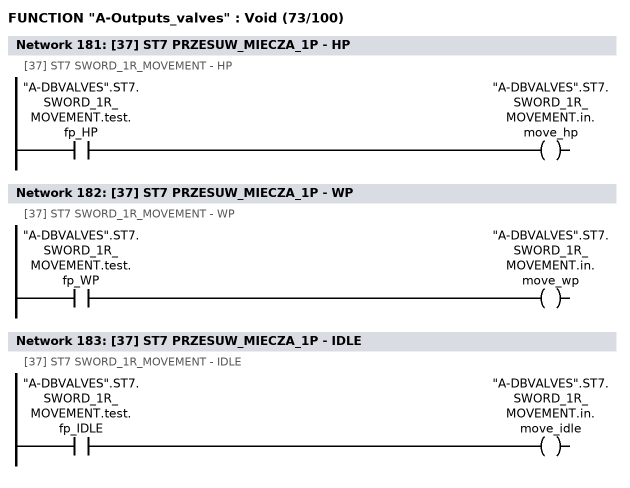
      O "A-DBVALVES".ST7.SWORD_1R_MOVEMENT.test.fp_HP;
//    O     "A-Flags".STATION.IN_HP_STEP
      = "A-DBVALVES".ST7.SWORD_1R_MOVEMENT.in.move_hp;
NETWORK
TITLE = [37] ST7 PRZESUW_MIECZA_1P - WP
//[37] ST7 SWORD_1R_MOVEMENT - WP
      O "A-DBVALVES".ST7.SWORD_1R_MOVEMENT.test.fp_WP;
      = "A-DBVALVES".ST7.SWORD_1R_MOVEMENT.in.move_wp;
NETWORK
TITLE = [37] ST7 PRZESUW_MIECZA_1P - IDLE
//[37] ST7 SWORD_1R_MOVEMENT - IDLE
      O "A-DBVALVES".ST7.SWORD_1R_MOVEMENT.test.fp_IDLE;
      = "A-DBVALVES".ST7.SWORD_1R_MOVEMENT.in.move_idle;
NETWORK
TITLE = [37] ST7 PRZESUW_MIECZA_1P
//[37] ST7 SWORD_1R_MOVEMENT
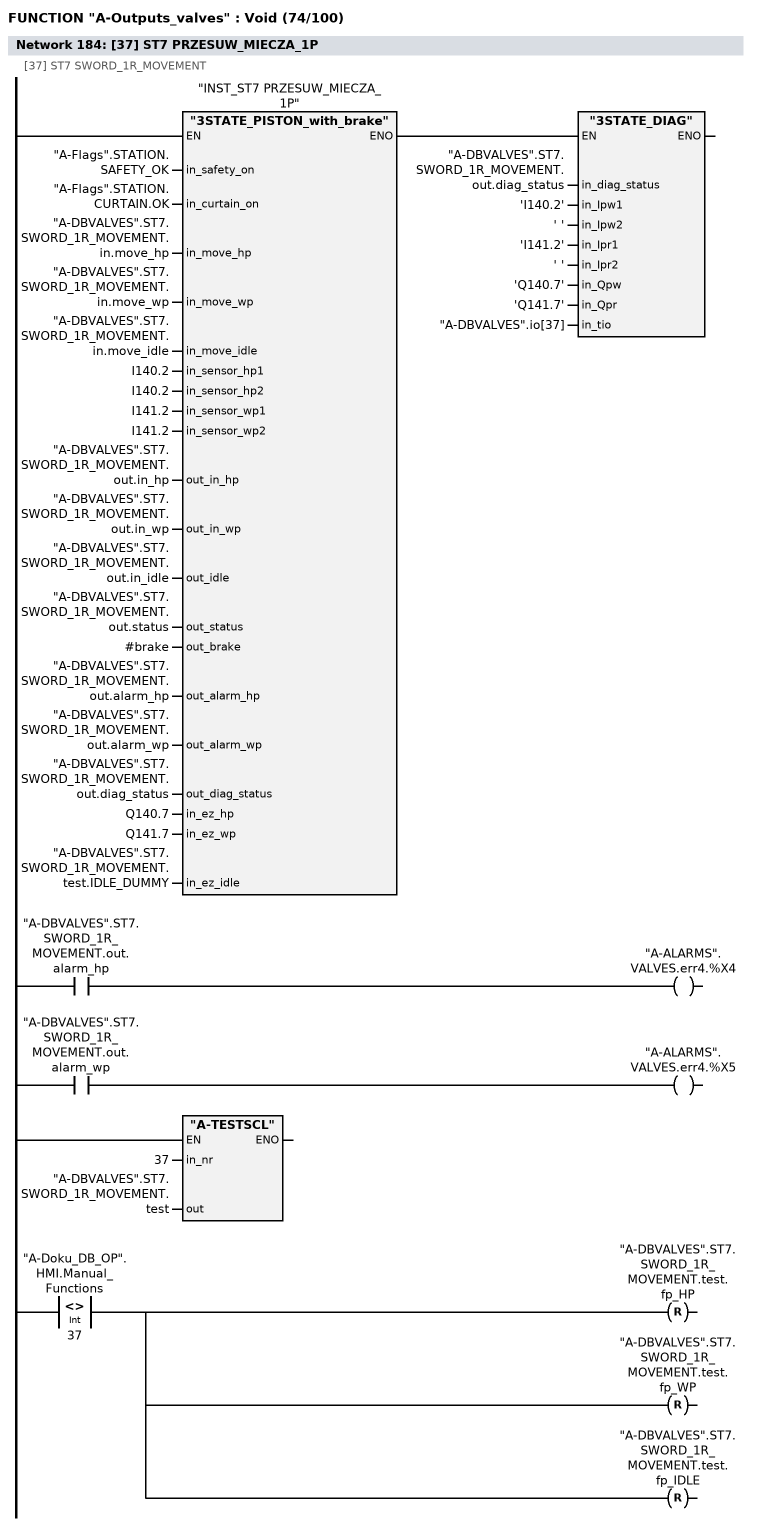
      CALL "3STATE_PISTON_with_brake", "INST_ST7 PRZESUW_MIECZA_1P"
      (  in_safety_on                := "A-Flags".STATION.SAFETY_OK ,
         in_curtain_on               := "A-Flags".STATION.CURTAIN.OK ,
         in_move_hp                  := "A-DBVALVES".ST7.SWORD_1R_MOVEMENT.in.move_hp ,
         in_move_wp                  := "A-DBVALVES".ST7.SWORD_1R_MOVEMENT.in.move_wp ,
         in_move_idle                := "A-DBVALVES".ST7.SWORD_1R_MOVEMENT.in.move_idle ,
         in_sensor_hp1               := I140.2 ,
         in_sensor_hp2               := I140.2 ,
         in_sensor_wp1               := I141.2 ,
         in_sensor_wp2               := I141.2 ,
         out_in_hp                   := "A-DBVALVES".ST7.SWORD_1R_MOVEMENT.out.in_hp ,
         out_in_wp                   := "A-DBVALVES".ST7.SWORD_1R_MOVEMENT.out.in_wp ,
         out_idle                    := "A-DBVALVES".ST7.SWORD_1R_MOVEMENT.out.in_idle ,
         out_status                  := "A-DBVALVES".ST7.SWORD_1R_MOVEMENT.out.status ,
         out_brake                   := #brake ,
         out_alarm_hp                := "A-DBVALVES".ST7.SWORD_1R_MOVEMENT.out.alarm_hp ,
         out_alarm_wp                := "A-DBVALVES".ST7.SWORD_1R_MOVEMENT.out.alarm_wp ,
         out_diag_status             := "A-DBVALVES".ST7.SWORD_1R_MOVEMENT.out.diag_status ,
         in_ez_hp                    := Q140.7 ,
         in_ez_wp                    := Q141.7 ,
         in_ez_idle                  := "A-DBVALVES".ST7.SWORD_1R_MOVEMENT.test.IDLE_DUMMY
      );

      CALL "3STATE_DIAG"
      (  in_diag_status              := "A-DBVALVES".ST7.SWORD_1R_MOVEMENT.out.diag_status ,
         in_Ipw1                     := 'I140.2' ,
         in_Ipw2                     := ' ' ,
         in_Ipr1                     := 'I141.2' ,
         in_Ipr2                     := ' ' ,
         in_Qpw                      := 'Q140.7' ,
         in_Qpr                      := 'Q141.7' ,
         in_tio                      := "A-DBVALVES".io[37]
      );

      A "A-DBVALVES".ST7.SWORD_1R_MOVEMENT.out.alarm_hp;
      = "A-ALARMS".VALVES.err4.%X4;

      A "A-DBVALVES".ST7.SWORD_1R_MOVEMENT.out.alarm_wp;
      = "A-ALARMS".VALVES.err4.%X5;

      CALL "A-TESTSCL"
      (  in_nr                       := 37 ,
         out                         := "A-DBVALVES".ST7.SWORD_1R_MOVEMENT.test
      );

      A(;
      L "A-Doku_DB_OP".HMI.Manual_Functions;
      L 37;
      <>I;
      );
      R "A-DBVALVES".ST7.SWORD_1R_MOVEMENT.test.fp_HP;
      R "A-DBVALVES".ST7.SWORD_1R_MOVEMENT.test.fp_WP;
      R "A-DBVALVES".ST7.SWORD_1R_MOVEMENT.test.fp_IDLE;
NETWORK
TITLE = -

NETWORK
TITLE = [38] ST7 PRZESUW_DOCISKOW - HP
//[38] ST7 HOLDFAST_MOVEMENT - HP
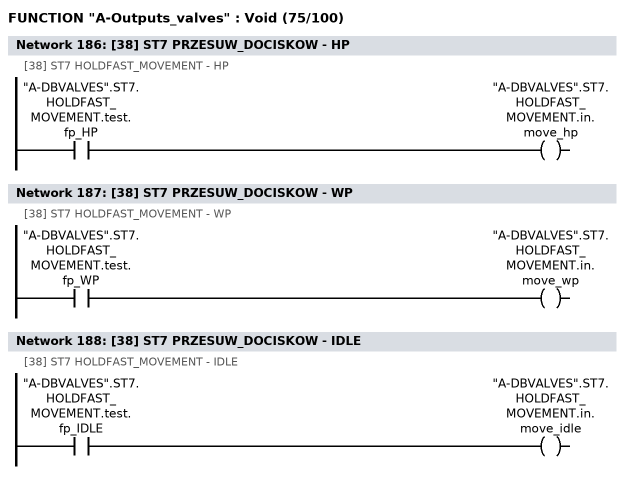
      O "A-DBVALVES".ST7.HOLDFAST_MOVEMENT.test.fp_HP;
//    O     "A-Flags".STATION.IN_HP_STEP
      = "A-DBVALVES".ST7.HOLDFAST_MOVEMENT.in.move_hp;
NETWORK
TITLE = [38] ST7 PRZESUW_DOCISKOW - WP
//[38] ST7 HOLDFAST_MOVEMENT - WP
      O "A-DBVALVES".ST7.HOLDFAST_MOVEMENT.test.fp_WP;
      = "A-DBVALVES".ST7.HOLDFAST_MOVEMENT.in.move_wp;
NETWORK
TITLE = [38] ST7 PRZESUW_DOCISKOW - IDLE
//[38] ST7 HOLDFAST_MOVEMENT - IDLE
      O "A-DBVALVES".ST7.HOLDFAST_MOVEMENT.test.fp_IDLE;
      = "A-DBVALVES".ST7.HOLDFAST_MOVEMENT.in.move_idle;
NETWORK
TITLE = [38] ST7 PRZESUW_DOCISKOW
//[38] ST7 HOLDFAST_MOVEMENT
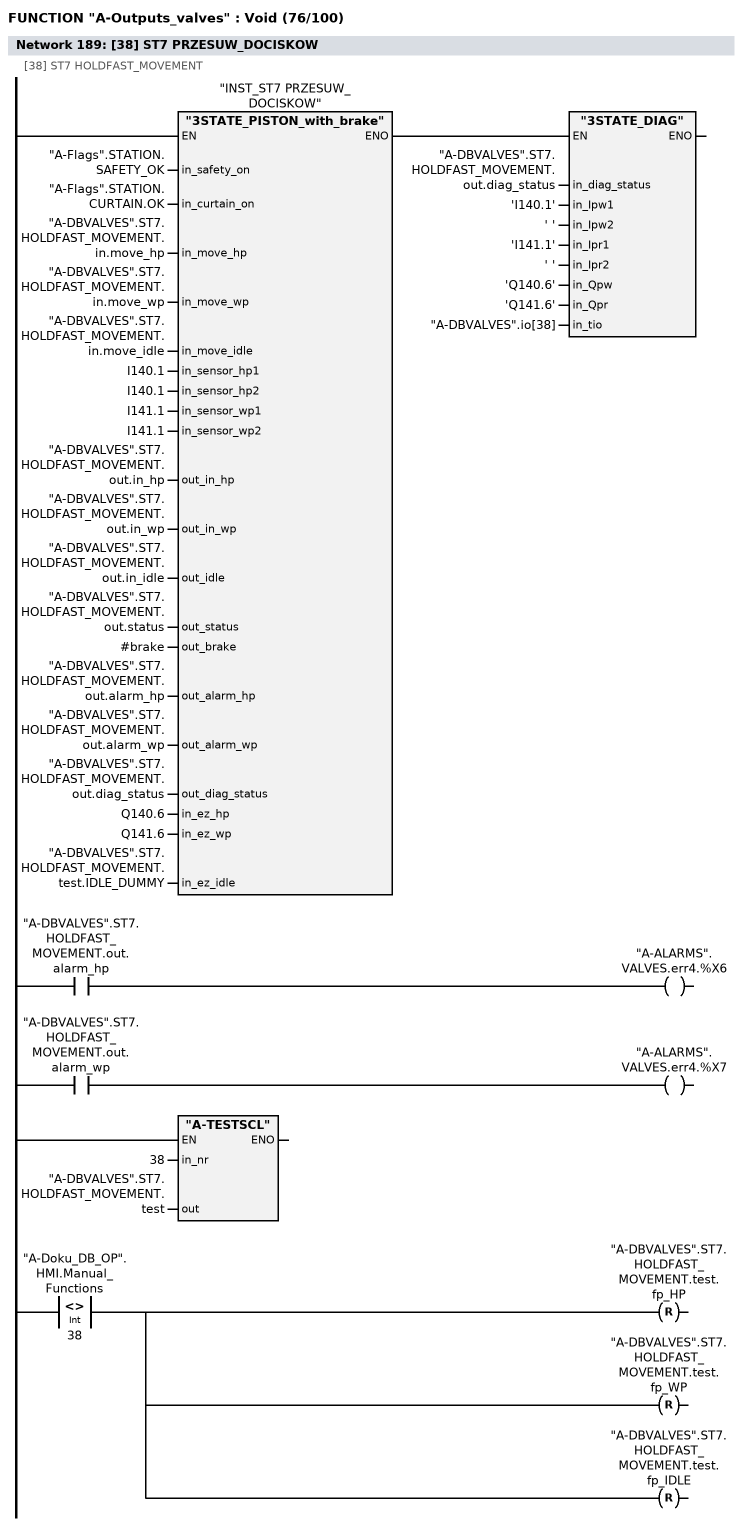
      CALL "3STATE_PISTON_with_brake", "INST_ST7 PRZESUW_DOCISKOW"
      (  in_safety_on                := "A-Flags".STATION.SAFETY_OK ,
         in_curtain_on               := "A-Flags".STATION.CURTAIN.OK ,
         in_move_hp                  := "A-DBVALVES".ST7.HOLDFAST_MOVEMENT.in.move_hp ,
         in_move_wp                  := "A-DBVALVES".ST7.HOLDFAST_MOVEMENT.in.move_wp ,
         in_move_idle                := "A-DBVALVES".ST7.HOLDFAST_MOVEMENT.in.move_idle ,
         in_sensor_hp1               := I140.1 ,
         in_sensor_hp2               := I140.1 ,
         in_sensor_wp1               := I141.1 ,
         in_sensor_wp2               := I141.1 ,
         out_in_hp                   := "A-DBVALVES".ST7.HOLDFAST_MOVEMENT.out.in_hp ,
         out_in_wp                   := "A-DBVALVES".ST7.HOLDFAST_MOVEMENT.out.in_wp ,
         out_idle                    := "A-DBVALVES".ST7.HOLDFAST_MOVEMENT.out.in_idle ,
         out_status                  := "A-DBVALVES".ST7.HOLDFAST_MOVEMENT.out.status ,
         out_brake                   := #brake ,
         out_alarm_hp                := "A-DBVALVES".ST7.HOLDFAST_MOVEMENT.out.alarm_hp ,
         out_alarm_wp                := "A-DBVALVES".ST7.HOLDFAST_MOVEMENT.out.alarm_wp ,
         out_diag_status             := "A-DBVALVES".ST7.HOLDFAST_MOVEMENT.out.diag_status ,
         in_ez_hp                    := Q140.6 ,
         in_ez_wp                    := Q141.6 ,
         in_ez_idle                  := "A-DBVALVES".ST7.HOLDFAST_MOVEMENT.test.IDLE_DUMMY
      );

      CALL "3STATE_DIAG"
      (  in_diag_status              := "A-DBVALVES".ST7.HOLDFAST_MOVEMENT.out.diag_status ,
         in_Ipw1                     := 'I140.1' ,
         in_Ipw2                     := ' ' ,
         in_Ipr1                     := 'I141.1' ,
         in_Ipr2                     := ' ' ,
         in_Qpw                      := 'Q140.6' ,
         in_Qpr                      := 'Q141.6' ,
         in_tio                      := "A-DBVALVES".io[38]
      );

      A "A-DBVALVES".ST7.HOLDFAST_MOVEMENT.out.alarm_hp;
      = "A-ALARMS".VALVES.err4.%X6;

      A "A-DBVALVES".ST7.HOLDFAST_MOVEMENT.out.alarm_wp;
      = "A-ALARMS".VALVES.err4.%X7;

      CALL "A-TESTSCL"
      (  in_nr                       := 38 ,
         out                         := "A-DBVALVES".ST7.HOLDFAST_MOVEMENT.test
      );

      A(;
      L "A-Doku_DB_OP".HMI.Manual_Functions;
      L 38;
      <>I;
      );
      R "A-DBVALVES".ST7.HOLDFAST_MOVEMENT.test.fp_HP;
      R "A-DBVALVES".ST7.HOLDFAST_MOVEMENT.test.fp_WP;
      R "A-DBVALVES".ST7.HOLDFAST_MOVEMENT.test.fp_IDLE;
NETWORK
TITLE = -

NETWORK
TITLE = [39] ST7 PRZESUW_MIECZA_Y_2L - HP
//[39] ST7 SWORD_Y_2L_MOVEMENT - HP
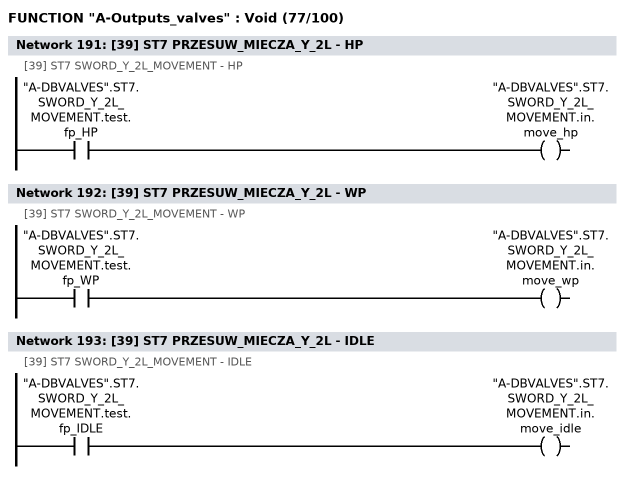
      O "A-DBVALVES".ST7.SWORD_Y_2L_MOVEMENT.test.fp_HP;
//    O     "A-Flags".STATION.IN_HP_STEP
      = "A-DBVALVES".ST7.SWORD_Y_2L_MOVEMENT.in.move_hp;
NETWORK
TITLE = [39] ST7 PRZESUW_MIECZA_Y_2L - WP
//[39] ST7 SWORD_Y_2L_MOVEMENT - WP
      O "A-DBVALVES".ST7.SWORD_Y_2L_MOVEMENT.test.fp_WP;
      = "A-DBVALVES".ST7.SWORD_Y_2L_MOVEMENT.in.move_wp;
NETWORK
TITLE = [39] ST7 PRZESUW_MIECZA_Y_2L - IDLE
//[39] ST7 SWORD_Y_2L_MOVEMENT - IDLE
      O "A-DBVALVES".ST7.SWORD_Y_2L_MOVEMENT.test.fp_IDLE;
      = "A-DBVALVES".ST7.SWORD_Y_2L_MOVEMENT.in.move_idle;
NETWORK
TITLE = [39] ST7 PRZESUW_MIECZA_Y_2L
//[39] ST7 SWORD_Y_2L_MOVEMENT
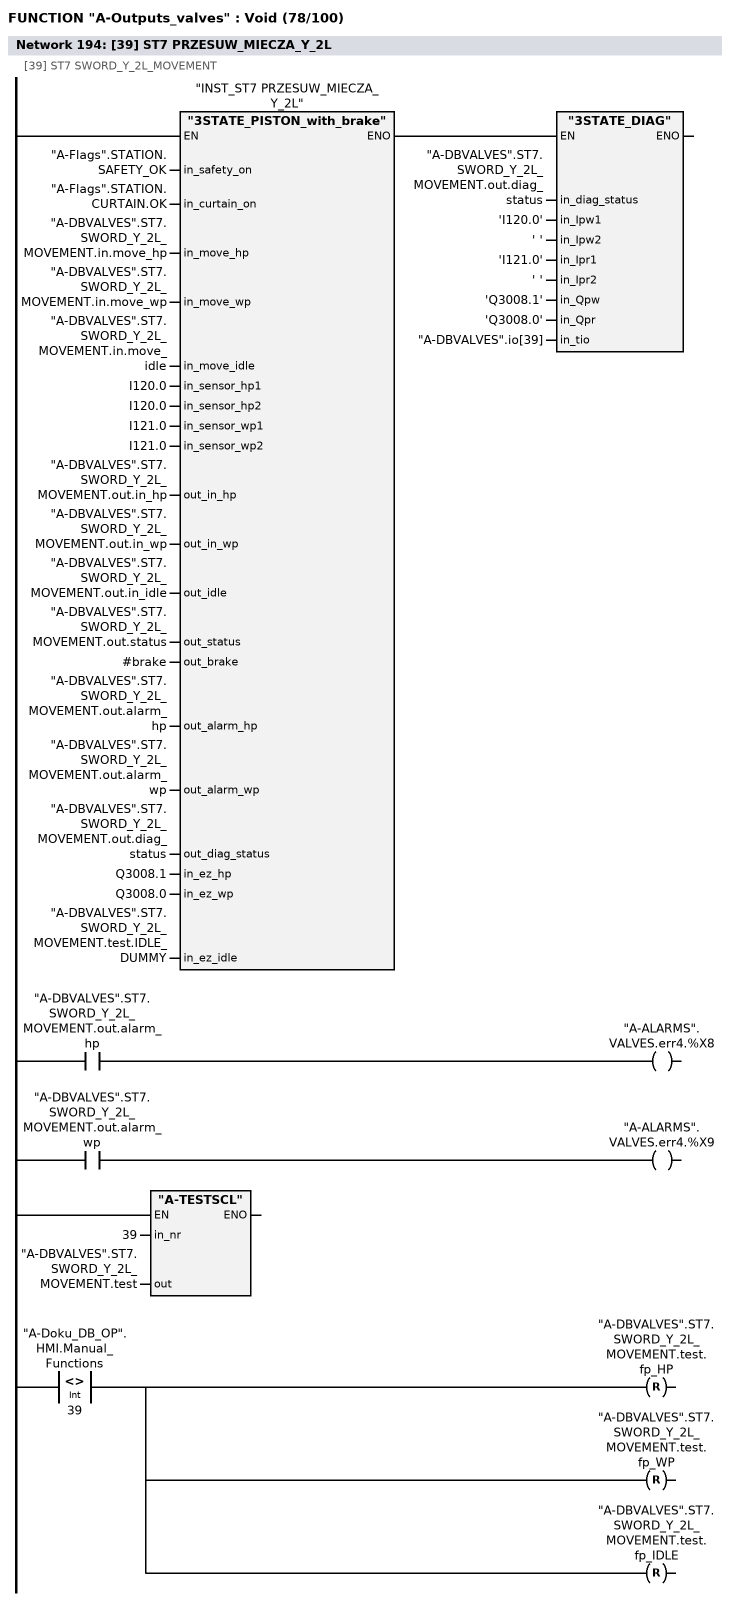
      CALL "3STATE_PISTON_with_brake", "INST_ST7 PRZESUW_MIECZA_Y_2L"
      (  in_safety_on                := "A-Flags".STATION.SAFETY_OK ,
         in_curtain_on               := "A-Flags".STATION.CURTAIN.OK ,
         in_move_hp                  := "A-DBVALVES".ST7.SWORD_Y_2L_MOVEMENT.in.move_hp ,
         in_move_wp                  := "A-DBVALVES".ST7.SWORD_Y_2L_MOVEMENT.in.move_wp ,
         in_move_idle                := "A-DBVALVES".ST7.SWORD_Y_2L_MOVEMENT.in.move_idle ,
         in_sensor_hp1               := I120.0 ,
         in_sensor_hp2               := I120.0 ,
         in_sensor_wp1               := I121.0 ,
         in_sensor_wp2               := I121.0 ,
         out_in_hp                   := "A-DBVALVES".ST7.SWORD_Y_2L_MOVEMENT.out.in_hp ,
         out_in_wp                   := "A-DBVALVES".ST7.SWORD_Y_2L_MOVEMENT.out.in_wp ,
         out_idle                    := "A-DBVALVES".ST7.SWORD_Y_2L_MOVEMENT.out.in_idle ,
         out_status                  := "A-DBVALVES".ST7.SWORD_Y_2L_MOVEMENT.out.status ,
         out_brake                   := #brake ,
         out_alarm_hp                := "A-DBVALVES".ST7.SWORD_Y_2L_MOVEMENT.out.alarm_hp ,
         out_alarm_wp                := "A-DBVALVES".ST7.SWORD_Y_2L_MOVEMENT.out.alarm_wp ,
         out_diag_status             := "A-DBVALVES".ST7.SWORD_Y_2L_MOVEMENT.out.diag_status ,
         in_ez_hp                    := Q3008.1 ,
         in_ez_wp                    := Q3008.0 ,
         in_ez_idle                  := "A-DBVALVES".ST7.SWORD_Y_2L_MOVEMENT.test.IDLE_DUMMY
      );

      CALL "3STATE_DIAG"
      (  in_diag_status              := "A-DBVALVES".ST7.SWORD_Y_2L_MOVEMENT.out.diag_status ,
         in_Ipw1                     := 'I120.0' ,
         in_Ipw2                     := ' ' ,
         in_Ipr1                     := 'I121.0' ,
         in_Ipr2                     := ' ' ,
         in_Qpw                      := 'Q3008.1' ,
         in_Qpr                      := 'Q3008.0' ,
         in_tio                      := "A-DBVALVES".io[39]
      );

      A "A-DBVALVES".ST7.SWORD_Y_2L_MOVEMENT.out.alarm_hp;
      = "A-ALARMS".VALVES.err4.%X8;

      A "A-DBVALVES".ST7.SWORD_Y_2L_MOVEMENT.out.alarm_wp;
      = "A-ALARMS".VALVES.err4.%X9;

      CALL "A-TESTSCL"
      (  in_nr                       := 39 ,
         out                         := "A-DBVALVES".ST7.SWORD_Y_2L_MOVEMENT.test
      );

      A(;
      L "A-Doku_DB_OP".HMI.Manual_Functions;
      L 39;
      <>I;
      );
      R "A-DBVALVES".ST7.SWORD_Y_2L_MOVEMENT.test.fp_HP;
      R "A-DBVALVES".ST7.SWORD_Y_2L_MOVEMENT.test.fp_WP;
      R "A-DBVALVES".ST7.SWORD_Y_2L_MOVEMENT.test.fp_IDLE;
NETWORK
TITLE = -

NETWORK
TITLE = [40] ST7 MIECZ_2L - HP
//[40] ST7 SWORD_2L - HP
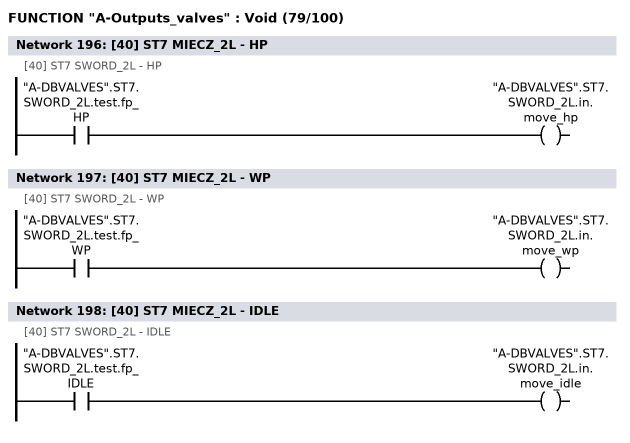
      O "A-DBVALVES".ST7.SWORD_2L.test.fp_HP;
//    O     "A-Flags".STATION.IN_HP_STEP
      = "A-DBVALVES".ST7.SWORD_2L.in.move_hp;
NETWORK
TITLE = [40] ST7 MIECZ_2L - WP
//[40] ST7 SWORD_2L - WP
      O "A-DBVALVES".ST7.SWORD_2L.test.fp_WP;
      = "A-DBVALVES".ST7.SWORD_2L.in.move_wp;
NETWORK
TITLE = [40] ST7 MIECZ_2L - IDLE
//[40] ST7 SWORD_2L - IDLE
      O "A-DBVALVES".ST7.SWORD_2L.test.fp_IDLE;
      = "A-DBVALVES".ST7.SWORD_2L.in.move_idle;
NETWORK
TITLE = [40] ST7 MIECZ_2L
//[40] ST7 SWORD_2L
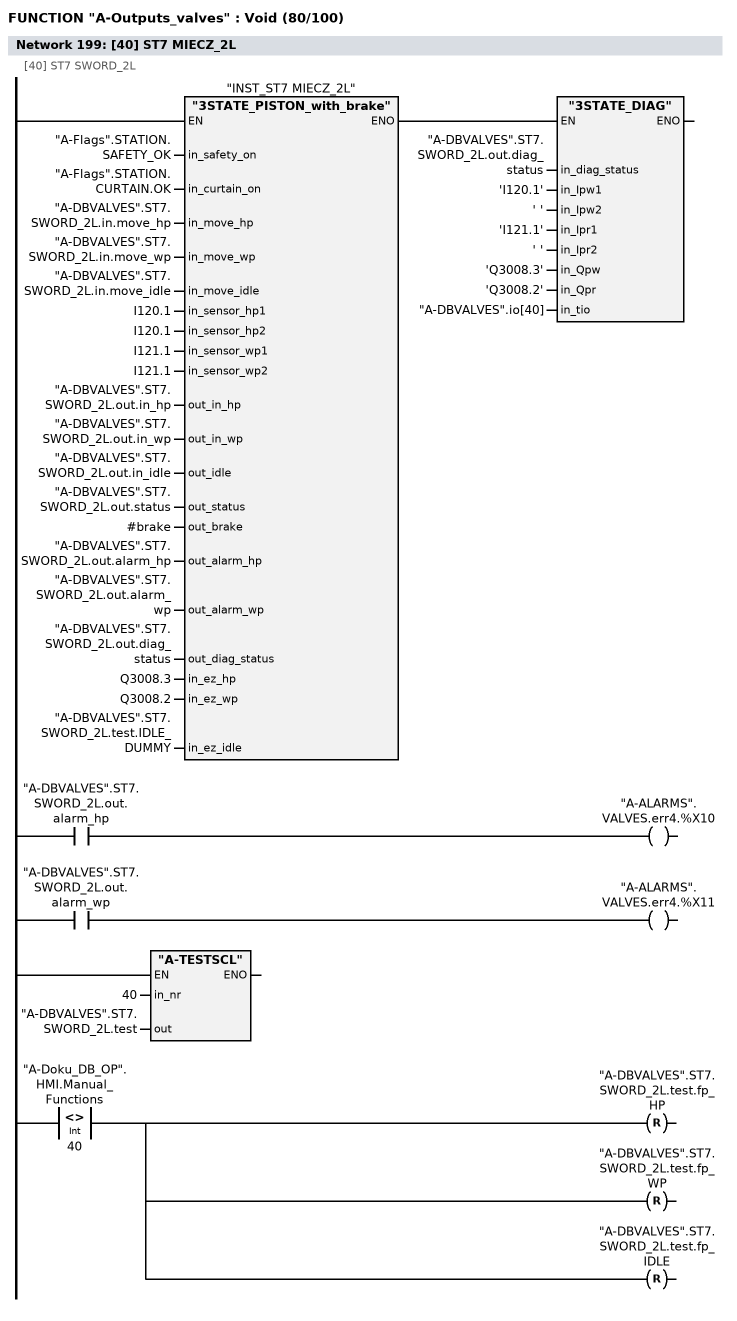
      CALL "3STATE_PISTON_with_brake", "INST_ST7 MIECZ_2L"
      (  in_safety_on                := "A-Flags".STATION.SAFETY_OK ,
         in_curtain_on               := "A-Flags".STATION.CURTAIN.OK ,
         in_move_hp                  := "A-DBVALVES".ST7.SWORD_2L.in.move_hp ,
         in_move_wp                  := "A-DBVALVES".ST7.SWORD_2L.in.move_wp ,
         in_move_idle                := "A-DBVALVES".ST7.SWORD_2L.in.move_idle ,
         in_sensor_hp1               := I120.1 ,
         in_sensor_hp2               := I120.1 ,
         in_sensor_wp1               := I121.1 ,
         in_sensor_wp2               := I121.1 ,
         out_in_hp                   := "A-DBVALVES".ST7.SWORD_2L.out.in_hp ,
         out_in_wp                   := "A-DBVALVES".ST7.SWORD_2L.out.in_wp ,
         out_idle                    := "A-DBVALVES".ST7.SWORD_2L.out.in_idle ,
         out_status                  := "A-DBVALVES".ST7.SWORD_2L.out.status ,
         out_brake                   := #brake ,
         out_alarm_hp                := "A-DBVALVES".ST7.SWORD_2L.out.alarm_hp ,
         out_alarm_wp                := "A-DBVALVES".ST7.SWORD_2L.out.alarm_wp ,
         out_diag_status             := "A-DBVALVES".ST7.SWORD_2L.out.diag_status ,
         in_ez_hp                    := Q3008.3 ,
         in_ez_wp                    := Q3008.2 ,
         in_ez_idle                  := "A-DBVALVES".ST7.SWORD_2L.test.IDLE_DUMMY
      );

      CALL "3STATE_DIAG"
      (  in_diag_status              := "A-DBVALVES".ST7.SWORD_2L.out.diag_status ,
         in_Ipw1                     := 'I120.1' ,
         in_Ipw2                     := ' ' ,
         in_Ipr1                     := 'I121.1' ,
         in_Ipr2                     := ' ' ,
         in_Qpw                      := 'Q3008.3' ,
         in_Qpr                      := 'Q3008.2' ,
         in_tio                      := "A-DBVALVES".io[40]
      );

      A "A-DBVALVES".ST7.SWORD_2L.out.alarm_hp;
      = "A-ALARMS".VALVES.err4.%X10;

      A "A-DBVALVES".ST7.SWORD_2L.out.alarm_wp;
      = "A-ALARMS".VALVES.err4.%X11;

      CALL "A-TESTSCL"
      (  in_nr                       := 40 ,
         out                         := "A-DBVALVES".ST7.SWORD_2L.test
      );

      A(;
      L "A-Doku_DB_OP".HMI.Manual_Functions;
      L 40;
      <>I;
      );
      R "A-DBVALVES".ST7.SWORD_2L.test.fp_HP;
      R "A-DBVALVES".ST7.SWORD_2L.test.fp_WP;
      R "A-DBVALVES".ST7.SWORD_2L.test.fp_IDLE;
NETWORK
TITLE = -

NETWORK
TITLE = [41] ST7 PRZESUW_MIECZA_Y_2P - HP
//[41] ST7 SWORD_Y_2R_MOVEMENT - HP
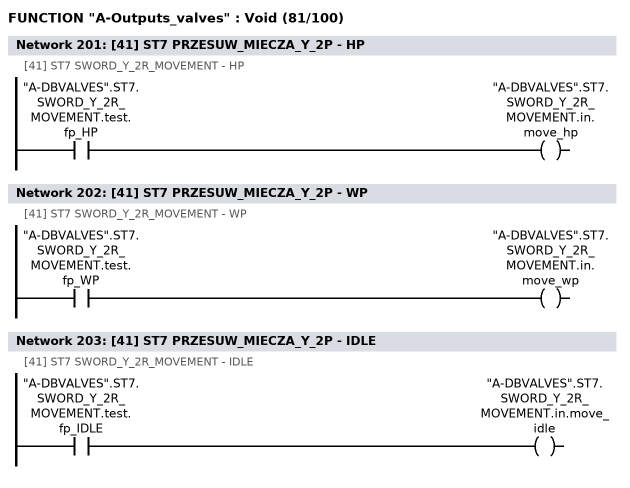
      O "A-DBVALVES".ST7.SWORD_Y_2R_MOVEMENT.test.fp_HP;
//    O     "A-Flags".STATION.IN_HP_STEP
      = "A-DBVALVES".ST7.SWORD_Y_2R_MOVEMENT.in.move_hp;
NETWORK
TITLE = [41] ST7 PRZESUW_MIECZA_Y_2P - WP
//[41] ST7 SWORD_Y_2R_MOVEMENT - WP
      O "A-DBVALVES".ST7.SWORD_Y_2R_MOVEMENT.test.fp_WP;
      = "A-DBVALVES".ST7.SWORD_Y_2R_MOVEMENT.in.move_wp;
NETWORK
TITLE = [41] ST7 PRZESUW_MIECZA_Y_2P - IDLE
//[41] ST7 SWORD_Y_2R_MOVEMENT - IDLE
      O "A-DBVALVES".ST7.SWORD_Y_2R_MOVEMENT.test.fp_IDLE;
      = "A-DBVALVES".ST7.SWORD_Y_2R_MOVEMENT.in.move_idle;
NETWORK
TITLE = [41] ST7 PRZESUW_MIECZA_Y_2P
//[41] ST7 SWORD_Y_2R_MOVEMENT
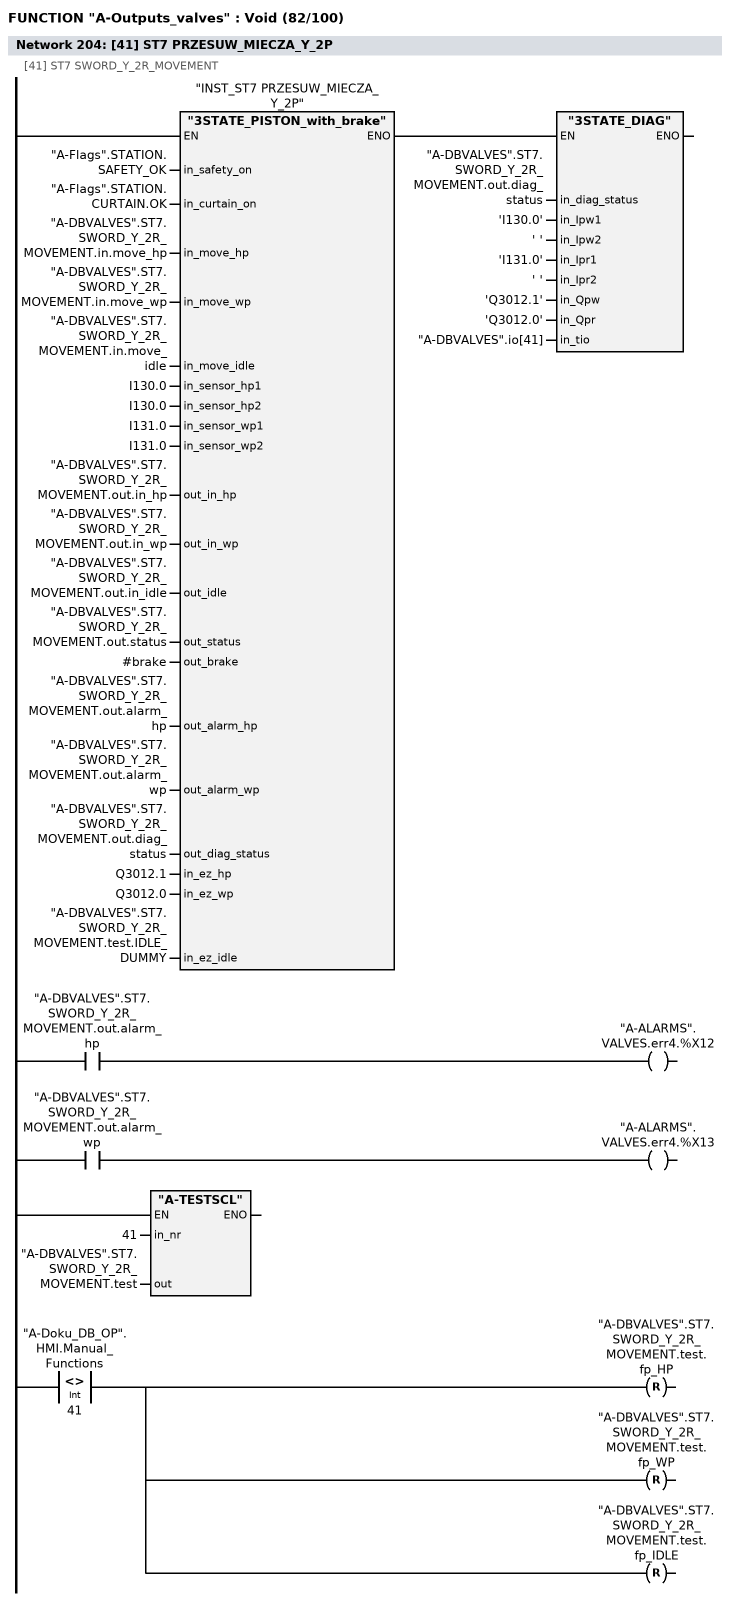
      CALL "3STATE_PISTON_with_brake", "INST_ST7 PRZESUW_MIECZA_Y_2P"
      (  in_safety_on                := "A-Flags".STATION.SAFETY_OK ,
         in_curtain_on               := "A-Flags".STATION.CURTAIN.OK ,
         in_move_hp                  := "A-DBVALVES".ST7.SWORD_Y_2R_MOVEMENT.in.move_hp ,
         in_move_wp                  := "A-DBVALVES".ST7.SWORD_Y_2R_MOVEMENT.in.move_wp ,
         in_move_idle                := "A-DBVALVES".ST7.SWORD_Y_2R_MOVEMENT.in.move_idle ,
         in_sensor_hp1               := I130.0 ,
         in_sensor_hp2               := I130.0 ,
         in_sensor_wp1               := I131.0 ,
         in_sensor_wp2               := I131.0 ,
         out_in_hp                   := "A-DBVALVES".ST7.SWORD_Y_2R_MOVEMENT.out.in_hp ,
         out_in_wp                   := "A-DBVALVES".ST7.SWORD_Y_2R_MOVEMENT.out.in_wp ,
         out_idle                    := "A-DBVALVES".ST7.SWORD_Y_2R_MOVEMENT.out.in_idle ,
         out_status                  := "A-DBVALVES".ST7.SWORD_Y_2R_MOVEMENT.out.status ,
         out_brake                   := #brake ,
         out_alarm_hp                := "A-DBVALVES".ST7.SWORD_Y_2R_MOVEMENT.out.alarm_hp ,
         out_alarm_wp                := "A-DBVALVES".ST7.SWORD_Y_2R_MOVEMENT.out.alarm_wp ,
         out_diag_status             := "A-DBVALVES".ST7.SWORD_Y_2R_MOVEMENT.out.diag_status ,
         in_ez_hp                    := Q3012.1 ,
         in_ez_wp                    := Q3012.0 ,
         in_ez_idle                  := "A-DBVALVES".ST7.SWORD_Y_2R_MOVEMENT.test.IDLE_DUMMY
      );

      CALL "3STATE_DIAG"
      (  in_diag_status              := "A-DBVALVES".ST7.SWORD_Y_2R_MOVEMENT.out.diag_status ,
         in_Ipw1                     := 'I130.0' ,
         in_Ipw2                     := ' ' ,
         in_Ipr1                     := 'I131.0' ,
         in_Ipr2                     := ' ' ,
         in_Qpw                      := 'Q3012.1' ,
         in_Qpr                      := 'Q3012.0' ,
         in_tio                      := "A-DBVALVES".io[41]
      );

      A "A-DBVALVES".ST7.SWORD_Y_2R_MOVEMENT.out.alarm_hp;
      = "A-ALARMS".VALVES.err4.%X12;

      A "A-DBVALVES".ST7.SWORD_Y_2R_MOVEMENT.out.alarm_wp;
      = "A-ALARMS".VALVES.err4.%X13;

      CALL "A-TESTSCL"
      (  in_nr                       := 41 ,
         out                         := "A-DBVALVES".ST7.SWORD_Y_2R_MOVEMENT.test
      );

      A(;
      L "A-Doku_DB_OP".HMI.Manual_Functions;
      L 41;
      <>I;
      );
      R "A-DBVALVES".ST7.SWORD_Y_2R_MOVEMENT.test.fp_HP;
      R "A-DBVALVES".ST7.SWORD_Y_2R_MOVEMENT.test.fp_WP;
      R "A-DBVALVES".ST7.SWORD_Y_2R_MOVEMENT.test.fp_IDLE;
NETWORK
TITLE = -

NETWORK
TITLE = [42] ST7 MIECZ_2P - HP
//[42] ST7 SWORD_2R - HP
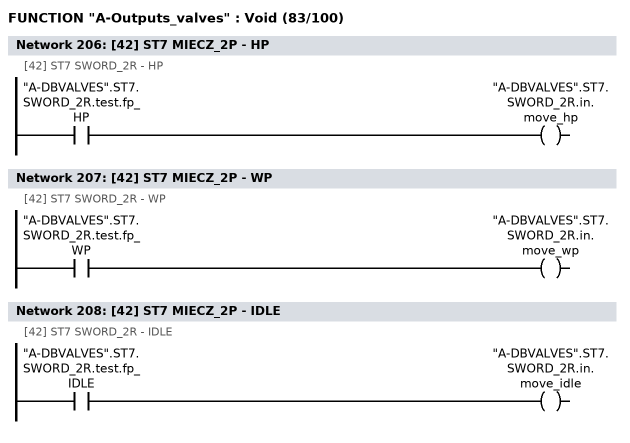
      O "A-DBVALVES".ST7.SWORD_2R.test.fp_HP;
//    O     "A-Flags".STATION.IN_HP_STEP
      = "A-DBVALVES".ST7.SWORD_2R.in.move_hp;
NETWORK
TITLE = [42] ST7 MIECZ_2P - WP
//[42] ST7 SWORD_2R - WP
      O "A-DBVALVES".ST7.SWORD_2R.test.fp_WP;
      = "A-DBVALVES".ST7.SWORD_2R.in.move_wp;
NETWORK
TITLE = [42] ST7 MIECZ_2P - IDLE
//[42] ST7 SWORD_2R - IDLE
      O "A-DBVALVES".ST7.SWORD_2R.test.fp_IDLE;
      = "A-DBVALVES".ST7.SWORD_2R.in.move_idle;
NETWORK
TITLE = [42] ST7 MIECZ_2P
//[42] ST7 SWORD_2R
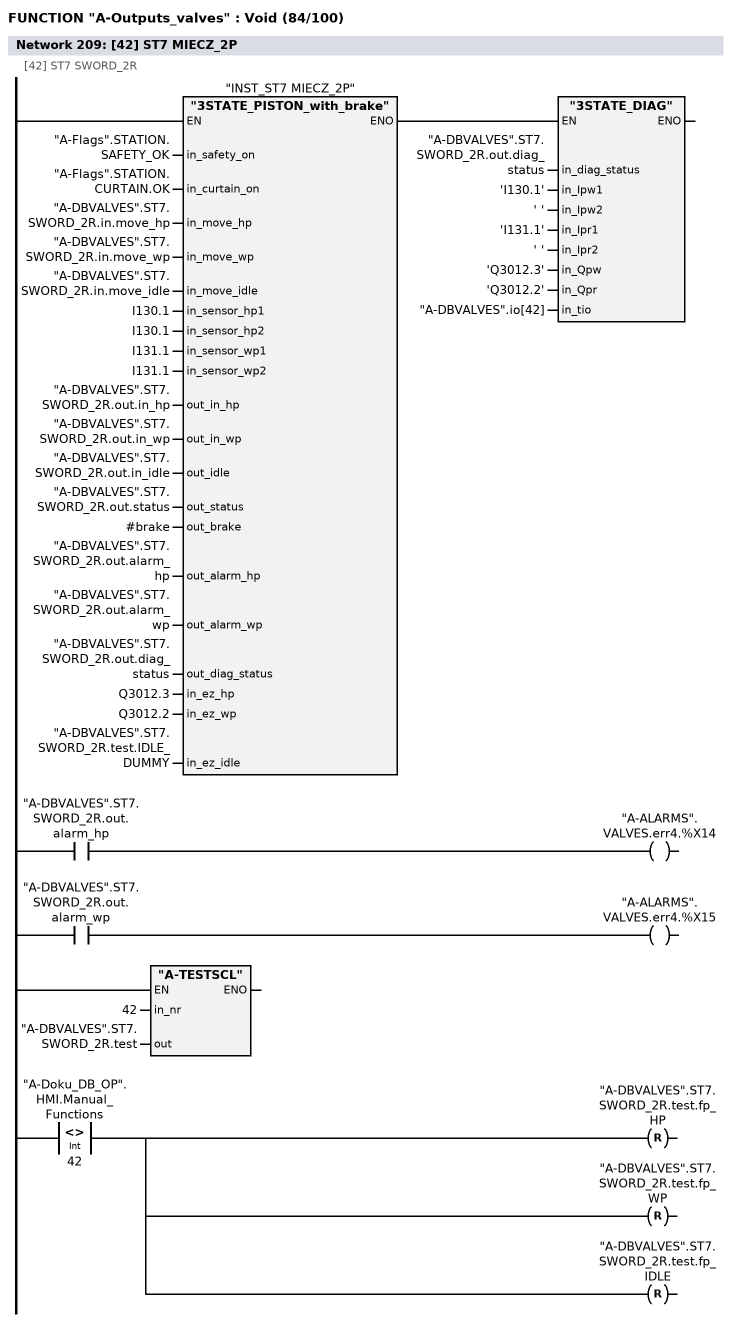
      CALL "3STATE_PISTON_with_brake", "INST_ST7 MIECZ_2P"
      (  in_safety_on                := "A-Flags".STATION.SAFETY_OK ,
         in_curtain_on               := "A-Flags".STATION.CURTAIN.OK ,
         in_move_hp                  := "A-DBVALVES".ST7.SWORD_2R.in.move_hp ,
         in_move_wp                  := "A-DBVALVES".ST7.SWORD_2R.in.move_wp ,
         in_move_idle                := "A-DBVALVES".ST7.SWORD_2R.in.move_idle ,
         in_sensor_hp1               := I130.1 ,
         in_sensor_hp2               := I130.1 ,
         in_sensor_wp1               := I131.1 ,
         in_sensor_wp2               := I131.1 ,
         out_in_hp                   := "A-DBVALVES".ST7.SWORD_2R.out.in_hp ,
         out_in_wp                   := "A-DBVALVES".ST7.SWORD_2R.out.in_wp ,
         out_idle                    := "A-DBVALVES".ST7.SWORD_2R.out.in_idle ,
         out_status                  := "A-DBVALVES".ST7.SWORD_2R.out.status ,
         out_brake                   := #brake ,
         out_alarm_hp                := "A-DBVALVES".ST7.SWORD_2R.out.alarm_hp ,
         out_alarm_wp                := "A-DBVALVES".ST7.SWORD_2R.out.alarm_wp ,
         out_diag_status             := "A-DBVALVES".ST7.SWORD_2R.out.diag_status ,
         in_ez_hp                    := Q3012.3 ,
         in_ez_wp                    := Q3012.2 ,
         in_ez_idle                  := "A-DBVALVES".ST7.SWORD_2R.test.IDLE_DUMMY
      );

      CALL "3STATE_DIAG"
      (  in_diag_status              := "A-DBVALVES".ST7.SWORD_2R.out.diag_status ,
         in_Ipw1                     := 'I130.1' ,
         in_Ipw2                     := ' ' ,
         in_Ipr1                     := 'I131.1' ,
         in_Ipr2                     := ' ' ,
         in_Qpw                      := 'Q3012.3' ,
         in_Qpr                      := 'Q3012.2' ,
         in_tio                      := "A-DBVALVES".io[42]
      );

      A "A-DBVALVES".ST7.SWORD_2R.out.alarm_hp;
      = "A-ALARMS".VALVES.err4.%X14;

      A "A-DBVALVES".ST7.SWORD_2R.out.alarm_wp;
      = "A-ALARMS".VALVES.err4.%X15;

      CALL "A-TESTSCL"
      (  in_nr                       := 42 ,
         out                         := "A-DBVALVES".ST7.SWORD_2R.test
      );

      A(;
      L "A-Doku_DB_OP".HMI.Manual_Functions;
      L 42;
      <>I;
      );
      R "A-DBVALVES".ST7.SWORD_2R.test.fp_HP;
      R "A-DBVALVES".ST7.SWORD_2R.test.fp_WP;
      R "A-DBVALVES".ST7.SWORD_2R.test.fp_IDLE;
NETWORK
TITLE = -

NETWORK
TITLE = [43] ST7 PRZESUW_MIECZA_X_3L - HP
//[43] ST7 SWORD_X_3L_MOVEMENT - HP
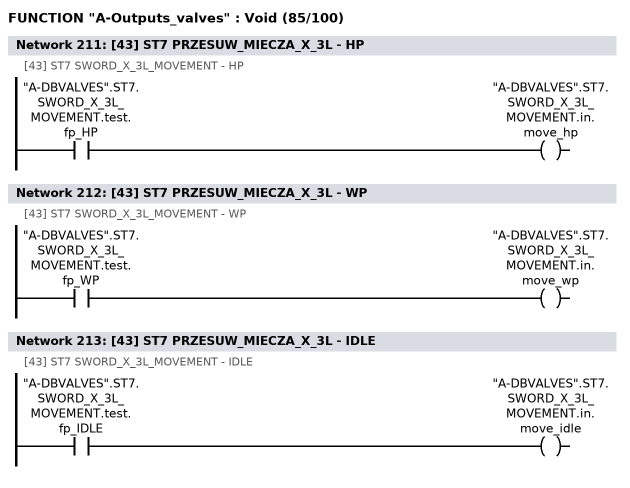
      O "A-DBVALVES".ST7.SWORD_X_3L_MOVEMENT.test.fp_HP;
//    O     "A-Flags".STATION.IN_HP_STEP
      = "A-DBVALVES".ST7.SWORD_X_3L_MOVEMENT.in.move_hp;
NETWORK
TITLE = [43] ST7 PRZESUW_MIECZA_X_3L - WP
//[43] ST7 SWORD_X_3L_MOVEMENT - WP
      O "A-DBVALVES".ST7.SWORD_X_3L_MOVEMENT.test.fp_WP;
      = "A-DBVALVES".ST7.SWORD_X_3L_MOVEMENT.in.move_wp;
NETWORK
TITLE = [43] ST7 PRZESUW_MIECZA_X_3L - IDLE
//[43] ST7 SWORD_X_3L_MOVEMENT - IDLE
      O "A-DBVALVES".ST7.SWORD_X_3L_MOVEMENT.test.fp_IDLE;
      = "A-DBVALVES".ST7.SWORD_X_3L_MOVEMENT.in.move_idle;
NETWORK
TITLE = [43] ST7 PRZESUW_MIECZA_X_3L
//[43] ST7 SWORD_X_3L_MOVEMENT
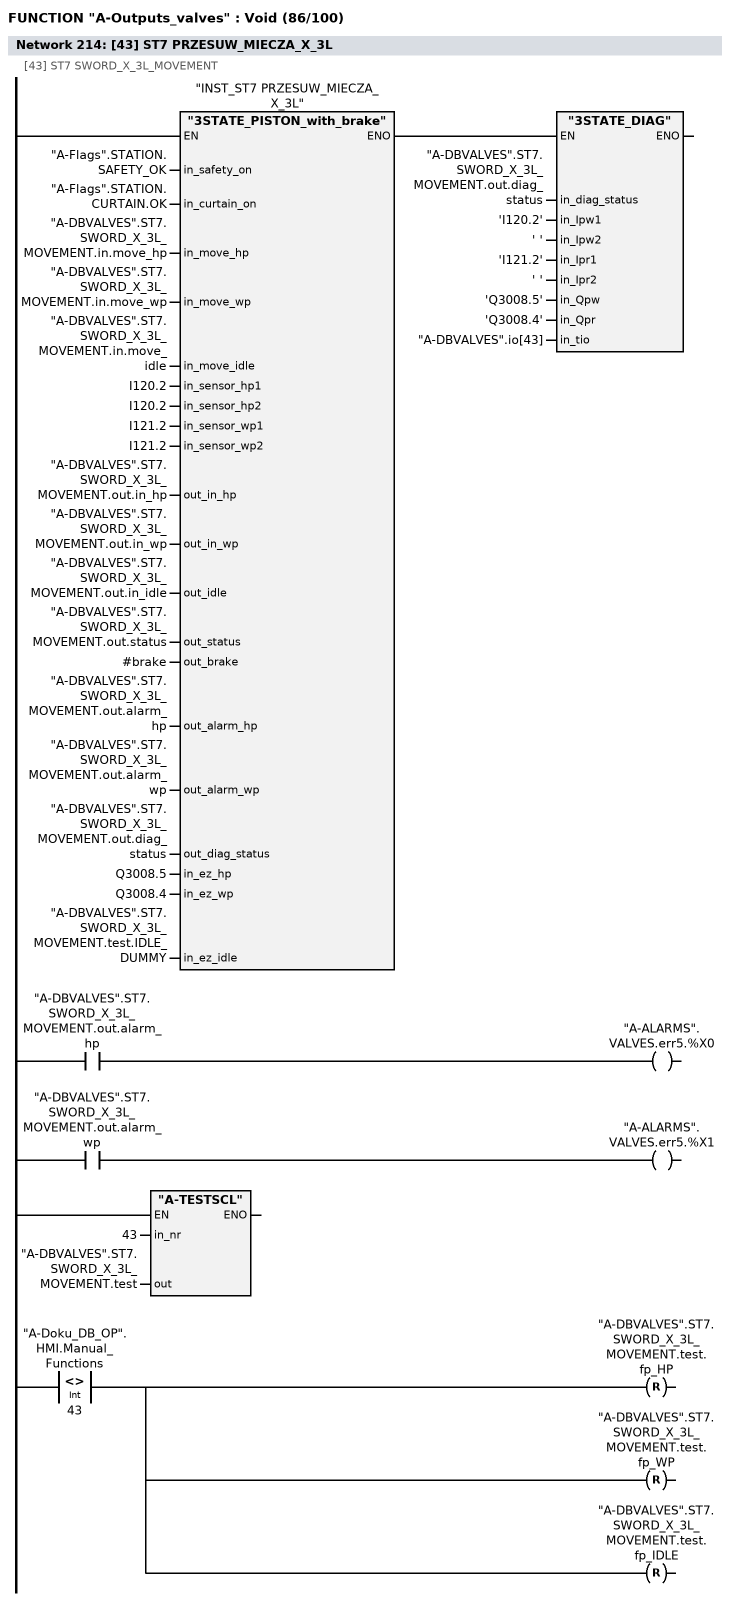
      CALL "3STATE_PISTON_with_brake", "INST_ST7 PRZESUW_MIECZA_X_3L"
      (  in_safety_on                := "A-Flags".STATION.SAFETY_OK ,
         in_curtain_on               := "A-Flags".STATION.CURTAIN.OK ,
         in_move_hp                  := "A-DBVALVES".ST7.SWORD_X_3L_MOVEMENT.in.move_hp ,
         in_move_wp                  := "A-DBVALVES".ST7.SWORD_X_3L_MOVEMENT.in.move_wp ,
         in_move_idle                := "A-DBVALVES".ST7.SWORD_X_3L_MOVEMENT.in.move_idle ,
         in_sensor_hp1               := I120.2 ,
         in_sensor_hp2               := I120.2 ,
         in_sensor_wp1               := I121.2 ,
         in_sensor_wp2               := I121.2 ,
         out_in_hp                   := "A-DBVALVES".ST7.SWORD_X_3L_MOVEMENT.out.in_hp ,
         out_in_wp                   := "A-DBVALVES".ST7.SWORD_X_3L_MOVEMENT.out.in_wp ,
         out_idle                    := "A-DBVALVES".ST7.SWORD_X_3L_MOVEMENT.out.in_idle ,
         out_status                  := "A-DBVALVES".ST7.SWORD_X_3L_MOVEMENT.out.status ,
         out_brake                   := #brake ,
         out_alarm_hp                := "A-DBVALVES".ST7.SWORD_X_3L_MOVEMENT.out.alarm_hp ,
         out_alarm_wp                := "A-DBVALVES".ST7.SWORD_X_3L_MOVEMENT.out.alarm_wp ,
         out_diag_status             := "A-DBVALVES".ST7.SWORD_X_3L_MOVEMENT.out.diag_status ,
         in_ez_hp                    := Q3008.5 ,
         in_ez_wp                    := Q3008.4 ,
         in_ez_idle                  := "A-DBVALVES".ST7.SWORD_X_3L_MOVEMENT.test.IDLE_DUMMY
      );

      CALL "3STATE_DIAG"
      (  in_diag_status              := "A-DBVALVES".ST7.SWORD_X_3L_MOVEMENT.out.diag_status ,
         in_Ipw1                     := 'I120.2' ,
         in_Ipw2                     := ' ' ,
         in_Ipr1                     := 'I121.2' ,
         in_Ipr2                     := ' ' ,
         in_Qpw                      := 'Q3008.5' ,
         in_Qpr                      := 'Q3008.4' ,
         in_tio                      := "A-DBVALVES".io[43]
      );

      A "A-DBVALVES".ST7.SWORD_X_3L_MOVEMENT.out.alarm_hp;
      = "A-ALARMS".VALVES.err5.%X0;

      A "A-DBVALVES".ST7.SWORD_X_3L_MOVEMENT.out.alarm_wp;
      = "A-ALARMS".VALVES.err5.%X1;

      CALL "A-TESTSCL"
      (  in_nr                       := 43 ,
         out                         := "A-DBVALVES".ST7.SWORD_X_3L_MOVEMENT.test
      );

      A(;
      L "A-Doku_DB_OP".HMI.Manual_Functions;
      L 43;
      <>I;
      );
      R "A-DBVALVES".ST7.SWORD_X_3L_MOVEMENT.test.fp_HP;
      R "A-DBVALVES".ST7.SWORD_X_3L_MOVEMENT.test.fp_WP;
      R "A-DBVALVES".ST7.SWORD_X_3L_MOVEMENT.test.fp_IDLE;
NETWORK
TITLE = -

NETWORK
TITLE = [44] ST7 PRZESUW_MIECZA_Y_3L - HP
//[44] ST7 SWORD_Y_3L_MOVEMENT - HP
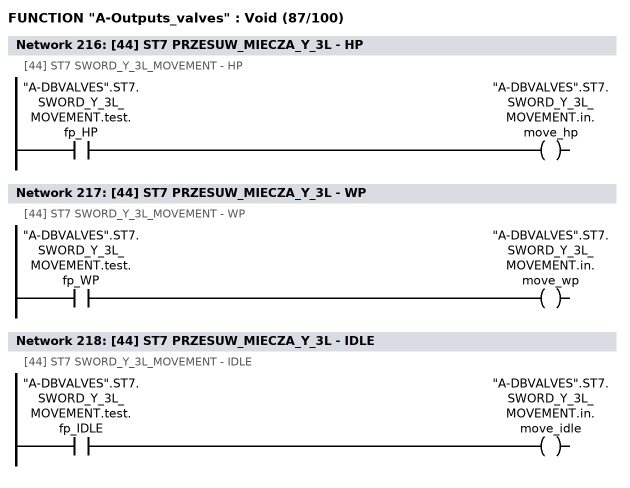
      O "A-DBVALVES".ST7.SWORD_Y_3L_MOVEMENT.test.fp_HP;
//    O     "A-Flags".STATION.IN_HP_STEP
      = "A-DBVALVES".ST7.SWORD_Y_3L_MOVEMENT.in.move_hp;
NETWORK
TITLE = [44] ST7 PRZESUW_MIECZA_Y_3L - WP
//[44] ST7 SWORD_Y_3L_MOVEMENT - WP
      O "A-DBVALVES".ST7.SWORD_Y_3L_MOVEMENT.test.fp_WP;
      = "A-DBVALVES".ST7.SWORD_Y_3L_MOVEMENT.in.move_wp;
NETWORK
TITLE = [44] ST7 PRZESUW_MIECZA_Y_3L - IDLE
//[44] ST7 SWORD_Y_3L_MOVEMENT - IDLE
      O "A-DBVALVES".ST7.SWORD_Y_3L_MOVEMENT.test.fp_IDLE;
      = "A-DBVALVES".ST7.SWORD_Y_3L_MOVEMENT.in.move_idle;
NETWORK
TITLE = [44] ST7 PRZESUW_MIECZA_Y_3L
//[44] ST7 SWORD_Y_3L_MOVEMENT
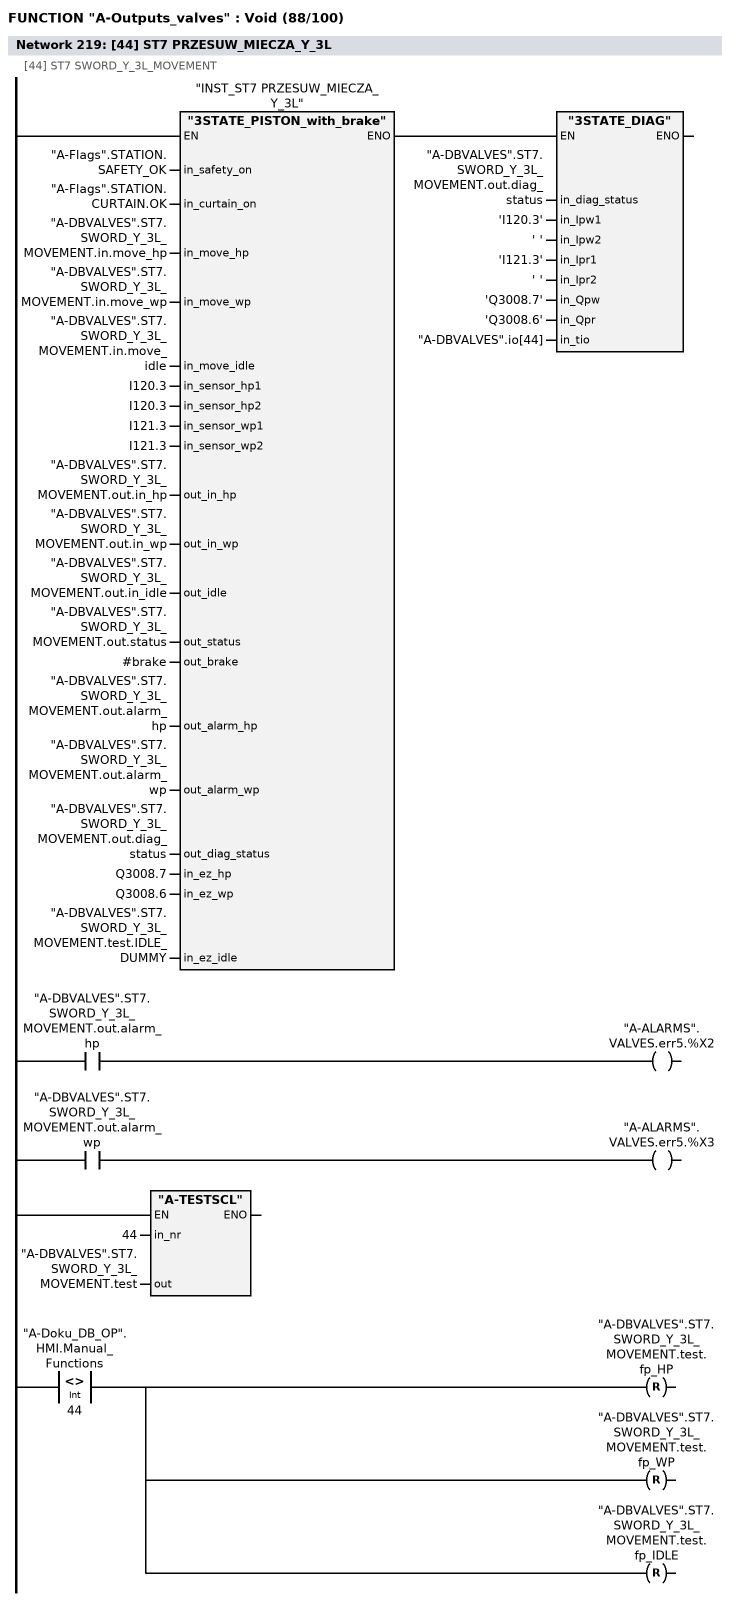
      CALL "3STATE_PISTON_with_brake", "INST_ST7 PRZESUW_MIECZA_Y_3L"
      (  in_safety_on                := "A-Flags".STATION.SAFETY_OK ,
         in_curtain_on               := "A-Flags".STATION.CURTAIN.OK ,
         in_move_hp                  := "A-DBVALVES".ST7.SWORD_Y_3L_MOVEMENT.in.move_hp ,
         in_move_wp                  := "A-DBVALVES".ST7.SWORD_Y_3L_MOVEMENT.in.move_wp ,
         in_move_idle                := "A-DBVALVES".ST7.SWORD_Y_3L_MOVEMENT.in.move_idle ,
         in_sensor_hp1               := I120.3 ,
         in_sensor_hp2               := I120.3 ,
         in_sensor_wp1               := I121.3 ,
         in_sensor_wp2               := I121.3 ,
         out_in_hp                   := "A-DBVALVES".ST7.SWORD_Y_3L_MOVEMENT.out.in_hp ,
         out_in_wp                   := "A-DBVALVES".ST7.SWORD_Y_3L_MOVEMENT.out.in_wp ,
         out_idle                    := "A-DBVALVES".ST7.SWORD_Y_3L_MOVEMENT.out.in_idle ,
         out_status                  := "A-DBVALVES".ST7.SWORD_Y_3L_MOVEMENT.out.status ,
         out_brake                   := #brake ,
         out_alarm_hp                := "A-DBVALVES".ST7.SWORD_Y_3L_MOVEMENT.out.alarm_hp ,
         out_alarm_wp                := "A-DBVALVES".ST7.SWORD_Y_3L_MOVEMENT.out.alarm_wp ,
         out_diag_status             := "A-DBVALVES".ST7.SWORD_Y_3L_MOVEMENT.out.diag_status ,
         in_ez_hp                    := Q3008.7 ,
         in_ez_wp                    := Q3008.6 ,
         in_ez_idle                  := "A-DBVALVES".ST7.SWORD_Y_3L_MOVEMENT.test.IDLE_DUMMY
      );

      CALL "3STATE_DIAG"
      (  in_diag_status              := "A-DBVALVES".ST7.SWORD_Y_3L_MOVEMENT.out.diag_status ,
         in_Ipw1                     := 'I120.3' ,
         in_Ipw2                     := ' ' ,
         in_Ipr1                     := 'I121.3' ,
         in_Ipr2                     := ' ' ,
         in_Qpw                      := 'Q3008.7' ,
         in_Qpr                      := 'Q3008.6' ,
         in_tio                      := "A-DBVALVES".io[44]
      );

      A "A-DBVALVES".ST7.SWORD_Y_3L_MOVEMENT.out.alarm_hp;
      = "A-ALARMS".VALVES.err5.%X2;

      A "A-DBVALVES".ST7.SWORD_Y_3L_MOVEMENT.out.alarm_wp;
      = "A-ALARMS".VALVES.err5.%X3;

      CALL "A-TESTSCL"
      (  in_nr                       := 44 ,
         out                         := "A-DBVALVES".ST7.SWORD_Y_3L_MOVEMENT.test
      );

      A(;
      L "A-Doku_DB_OP".HMI.Manual_Functions;
      L 44;
      <>I;
      );
      R "A-DBVALVES".ST7.SWORD_Y_3L_MOVEMENT.test.fp_HP;
      R "A-DBVALVES".ST7.SWORD_Y_3L_MOVEMENT.test.fp_WP;
      R "A-DBVALVES".ST7.SWORD_Y_3L_MOVEMENT.test.fp_IDLE;
NETWORK
TITLE = -

NETWORK
TITLE = [45] ST7 MIECZ_3L - HP
//[45] ST7 SWORD_3L - HP
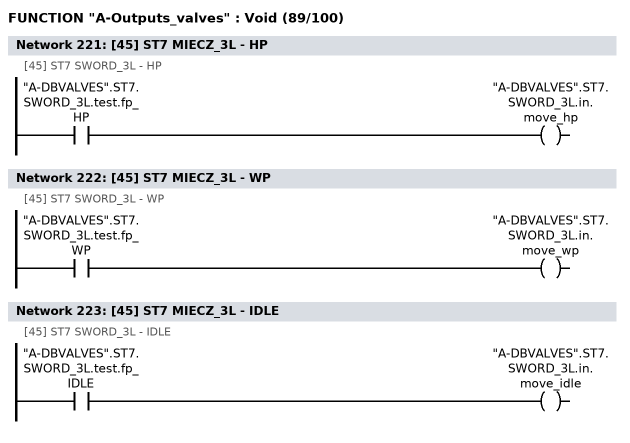
      O "A-DBVALVES".ST7.SWORD_3L.test.fp_HP;
//    O     "A-Flags".STATION.IN_HP_STEP
      = "A-DBVALVES".ST7.SWORD_3L.in.move_hp;
NETWORK
TITLE = [45] ST7 MIECZ_3L - WP
//[45] ST7 SWORD_3L - WP
      O "A-DBVALVES".ST7.SWORD_3L.test.fp_WP;
      = "A-DBVALVES".ST7.SWORD_3L.in.move_wp;
NETWORK
TITLE = [45] ST7 MIECZ_3L - IDLE
//[45] ST7 SWORD_3L - IDLE
      O "A-DBVALVES".ST7.SWORD_3L.test.fp_IDLE;
      = "A-DBVALVES".ST7.SWORD_3L.in.move_idle;
NETWORK
TITLE = [45] ST7 MIECZ_3L
//[45] ST7 SWORD_3L
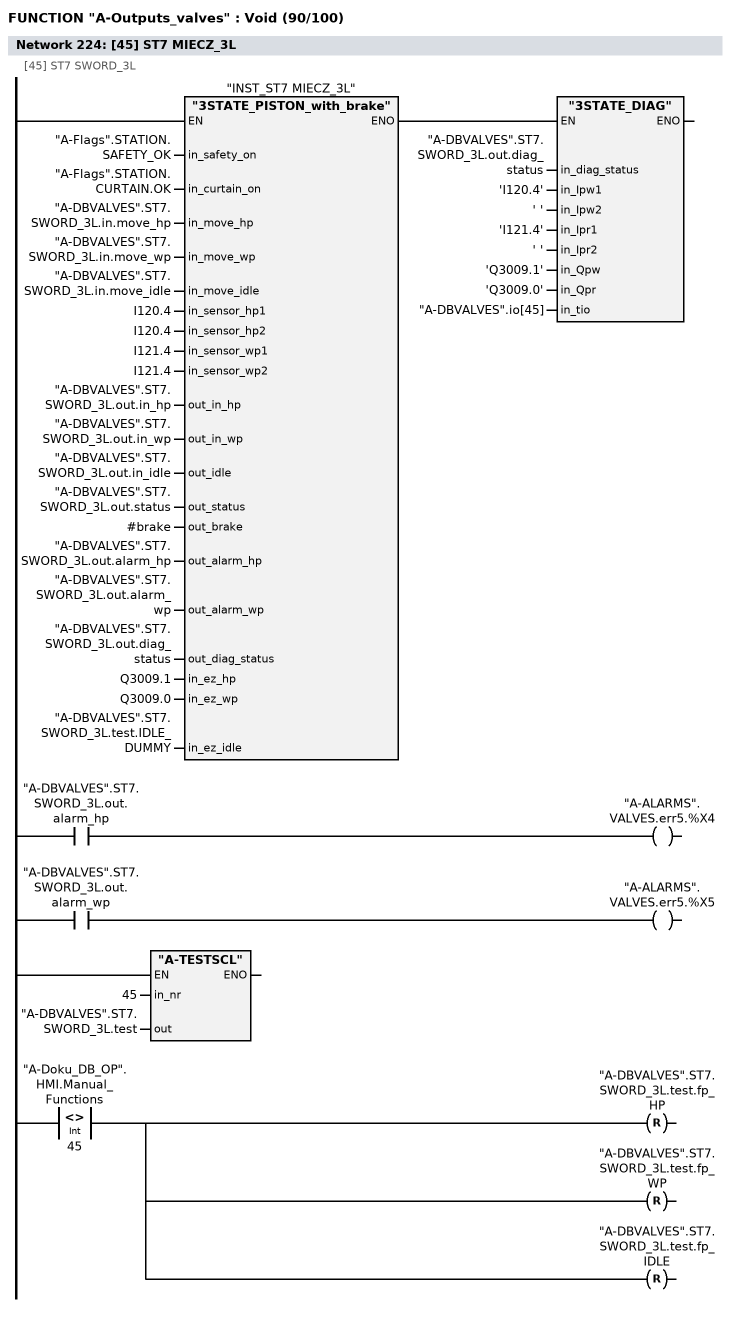
      CALL "3STATE_PISTON_with_brake", "INST_ST7 MIECZ_3L"
      (  in_safety_on                := "A-Flags".STATION.SAFETY_OK ,
         in_curtain_on               := "A-Flags".STATION.CURTAIN.OK ,
         in_move_hp                  := "A-DBVALVES".ST7.SWORD_3L.in.move_hp ,
         in_move_wp                  := "A-DBVALVES".ST7.SWORD_3L.in.move_wp ,
         in_move_idle                := "A-DBVALVES".ST7.SWORD_3L.in.move_idle ,
         in_sensor_hp1               := I120.4 ,
         in_sensor_hp2               := I120.4 ,
         in_sensor_wp1               := I121.4 ,
         in_sensor_wp2               := I121.4 ,
         out_in_hp                   := "A-DBVALVES".ST7.SWORD_3L.out.in_hp ,
         out_in_wp                   := "A-DBVALVES".ST7.SWORD_3L.out.in_wp ,
         out_idle                    := "A-DBVALVES".ST7.SWORD_3L.out.in_idle ,
         out_status                  := "A-DBVALVES".ST7.SWORD_3L.out.status ,
         out_brake                   := #brake ,
         out_alarm_hp                := "A-DBVALVES".ST7.SWORD_3L.out.alarm_hp ,
         out_alarm_wp                := "A-DBVALVES".ST7.SWORD_3L.out.alarm_wp ,
         out_diag_status             := "A-DBVALVES".ST7.SWORD_3L.out.diag_status ,
         in_ez_hp                    := Q3009.1 ,
         in_ez_wp                    := Q3009.0 ,
         in_ez_idle                  := "A-DBVALVES".ST7.SWORD_3L.test.IDLE_DUMMY
      );

      CALL "3STATE_DIAG"
      (  in_diag_status              := "A-DBVALVES".ST7.SWORD_3L.out.diag_status ,
         in_Ipw1                     := 'I120.4' ,
         in_Ipw2                     := ' ' ,
         in_Ipr1                     := 'I121.4' ,
         in_Ipr2                     := ' ' ,
         in_Qpw                      := 'Q3009.1' ,
         in_Qpr                      := 'Q3009.0' ,
         in_tio                      := "A-DBVALVES".io[45]
      );

      A "A-DBVALVES".ST7.SWORD_3L.out.alarm_hp;
      = "A-ALARMS".VALVES.err5.%X4;

      A "A-DBVALVES".ST7.SWORD_3L.out.alarm_wp;
      = "A-ALARMS".VALVES.err5.%X5;

      CALL "A-TESTSCL"
      (  in_nr                       := 45 ,
         out                         := "A-DBVALVES".ST7.SWORD_3L.test
      );

      A(;
      L "A-Doku_DB_OP".HMI.Manual_Functions;
      L 45;
      <>I;
      );
      R "A-DBVALVES".ST7.SWORD_3L.test.fp_HP;
      R "A-DBVALVES".ST7.SWORD_3L.test.fp_WP;
      R "A-DBVALVES".ST7.SWORD_3L.test.fp_IDLE;
NETWORK
TITLE = -

NETWORK
TITLE = [46] ST7 PRZESUW_MIECZA_X_3P - HP
//[46] ST7 SWORD_X_3R_MOVEMENT - HP
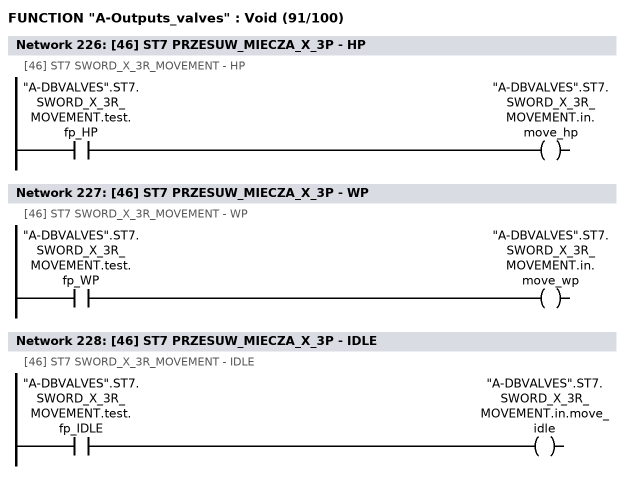
      O "A-DBVALVES".ST7.SWORD_X_3R_MOVEMENT.test.fp_HP;
//    O     "A-Flags".STATION.IN_HP_STEP
      = "A-DBVALVES".ST7.SWORD_X_3R_MOVEMENT.in.move_hp;
NETWORK
TITLE = [46] ST7 PRZESUW_MIECZA_X_3P - WP
//[46] ST7 SWORD_X_3R_MOVEMENT - WP
      O "A-DBVALVES".ST7.SWORD_X_3R_MOVEMENT.test.fp_WP;
      = "A-DBVALVES".ST7.SWORD_X_3R_MOVEMENT.in.move_wp;
NETWORK
TITLE = [46] ST7 PRZESUW_MIECZA_X_3P - IDLE
//[46] ST7 SWORD_X_3R_MOVEMENT - IDLE
      O "A-DBVALVES".ST7.SWORD_X_3R_MOVEMENT.test.fp_IDLE;
      = "A-DBVALVES".ST7.SWORD_X_3R_MOVEMENT.in.move_idle;
NETWORK
TITLE = [46] ST7 PRZESUW_MIECZA_X_3P
//[46] ST7 SWORD_X_3R_MOVEMENT
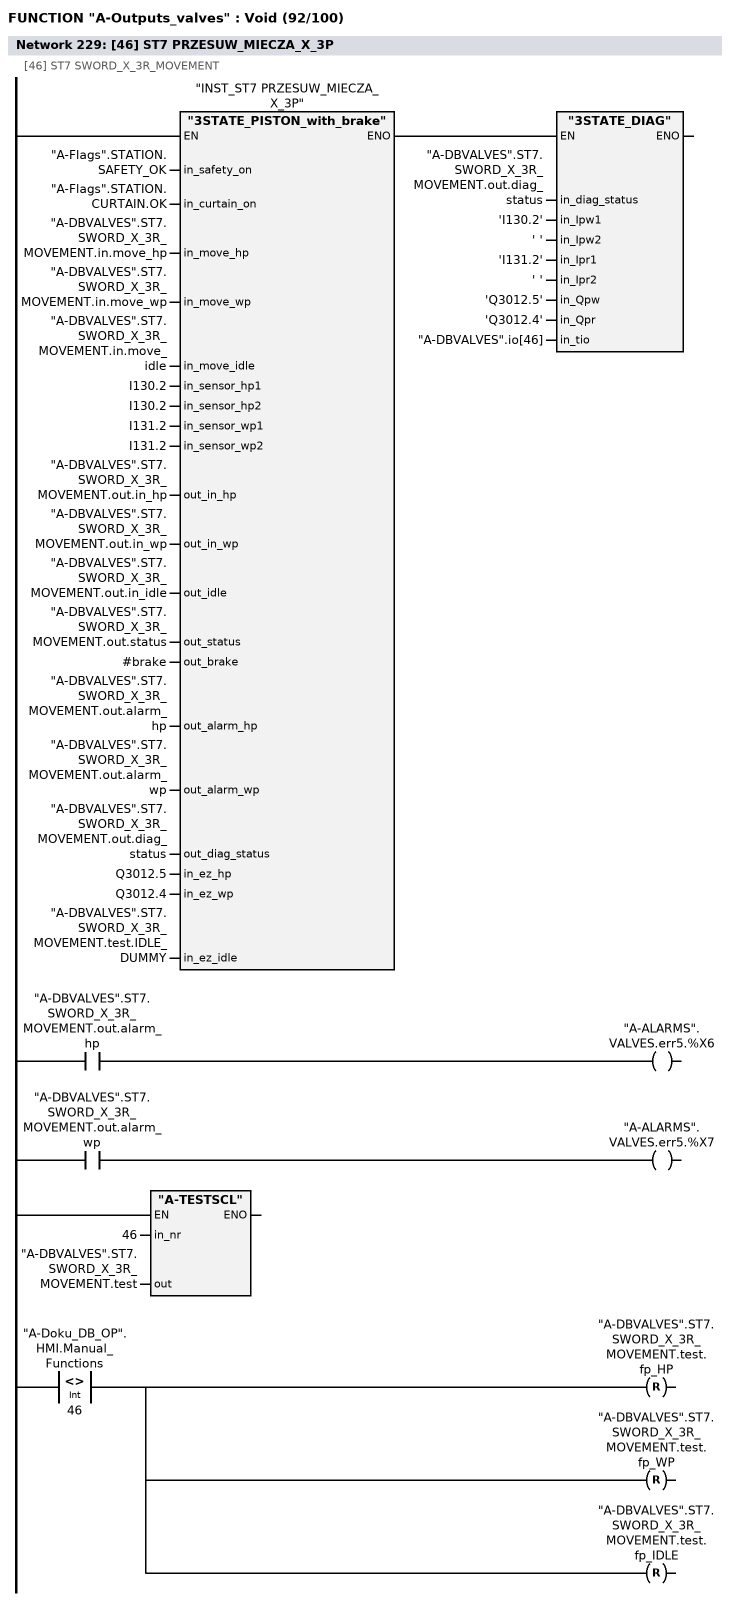
      CALL "3STATE_PISTON_with_brake", "INST_ST7 PRZESUW_MIECZA_X_3P"
      (  in_safety_on                := "A-Flags".STATION.SAFETY_OK ,
         in_curtain_on               := "A-Flags".STATION.CURTAIN.OK ,
         in_move_hp                  := "A-DBVALVES".ST7.SWORD_X_3R_MOVEMENT.in.move_hp ,
         in_move_wp                  := "A-DBVALVES".ST7.SWORD_X_3R_MOVEMENT.in.move_wp ,
         in_move_idle                := "A-DBVALVES".ST7.SWORD_X_3R_MOVEMENT.in.move_idle ,
         in_sensor_hp1               := I130.2 ,
         in_sensor_hp2               := I130.2 ,
         in_sensor_wp1               := I131.2 ,
         in_sensor_wp2               := I131.2 ,
         out_in_hp                   := "A-DBVALVES".ST7.SWORD_X_3R_MOVEMENT.out.in_hp ,
         out_in_wp                   := "A-DBVALVES".ST7.SWORD_X_3R_MOVEMENT.out.in_wp ,
         out_idle                    := "A-DBVALVES".ST7.SWORD_X_3R_MOVEMENT.out.in_idle ,
         out_status                  := "A-DBVALVES".ST7.SWORD_X_3R_MOVEMENT.out.status ,
         out_brake                   := #brake ,
         out_alarm_hp                := "A-DBVALVES".ST7.SWORD_X_3R_MOVEMENT.out.alarm_hp ,
         out_alarm_wp                := "A-DBVALVES".ST7.SWORD_X_3R_MOVEMENT.out.alarm_wp ,
         out_diag_status             := "A-DBVALVES".ST7.SWORD_X_3R_MOVEMENT.out.diag_status ,
         in_ez_hp                    := Q3012.5 ,
         in_ez_wp                    := Q3012.4 ,
         in_ez_idle                  := "A-DBVALVES".ST7.SWORD_X_3R_MOVEMENT.test.IDLE_DUMMY
      );

      CALL "3STATE_DIAG"
      (  in_diag_status              := "A-DBVALVES".ST7.SWORD_X_3R_MOVEMENT.out.diag_status ,
         in_Ipw1                     := 'I130.2' ,
         in_Ipw2                     := ' ' ,
         in_Ipr1                     := 'I131.2' ,
         in_Ipr2                     := ' ' ,
         in_Qpw                      := 'Q3012.5' ,
         in_Qpr                      := 'Q3012.4' ,
         in_tio                      := "A-DBVALVES".io[46]
      );

      A "A-DBVALVES".ST7.SWORD_X_3R_MOVEMENT.out.alarm_hp;
      = "A-ALARMS".VALVES.err5.%X6;

      A "A-DBVALVES".ST7.SWORD_X_3R_MOVEMENT.out.alarm_wp;
      = "A-ALARMS".VALVES.err5.%X7;

      CALL "A-TESTSCL"
      (  in_nr                       := 46 ,
         out                         := "A-DBVALVES".ST7.SWORD_X_3R_MOVEMENT.test
      );

      A(;
      L "A-Doku_DB_OP".HMI.Manual_Functions;
      L 46;
      <>I;
      );
      R "A-DBVALVES".ST7.SWORD_X_3R_MOVEMENT.test.fp_HP;
      R "A-DBVALVES".ST7.SWORD_X_3R_MOVEMENT.test.fp_WP;
      R "A-DBVALVES".ST7.SWORD_X_3R_MOVEMENT.test.fp_IDLE;
NETWORK
TITLE = -

NETWORK
TITLE = [47] ST7 PRZESUW_MIECZA_Y_3P - HP
//[47] ST7 SWORD_Y_3R_MOVEMENT - HP
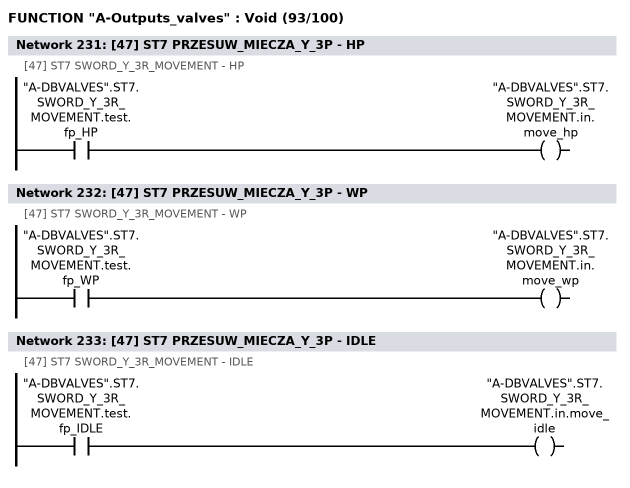
      O "A-DBVALVES".ST7.SWORD_Y_3R_MOVEMENT.test.fp_HP;
//    O     "A-Flags".STATION.IN_HP_STEP
      = "A-DBVALVES".ST7.SWORD_Y_3R_MOVEMENT.in.move_hp;
NETWORK
TITLE = [47] ST7 PRZESUW_MIECZA_Y_3P - WP
//[47] ST7 SWORD_Y_3R_MOVEMENT - WP
      O "A-DBVALVES".ST7.SWORD_Y_3R_MOVEMENT.test.fp_WP;
      = "A-DBVALVES".ST7.SWORD_Y_3R_MOVEMENT.in.move_wp;
NETWORK
TITLE = [47] ST7 PRZESUW_MIECZA_Y_3P - IDLE
//[47] ST7 SWORD_Y_3R_MOVEMENT - IDLE
      O "A-DBVALVES".ST7.SWORD_Y_3R_MOVEMENT.test.fp_IDLE;
      = "A-DBVALVES".ST7.SWORD_Y_3R_MOVEMENT.in.move_idle;
NETWORK
TITLE = [47] ST7 PRZESUW_MIECZA_Y_3P
//[47] ST7 SWORD_Y_3R_MOVEMENT
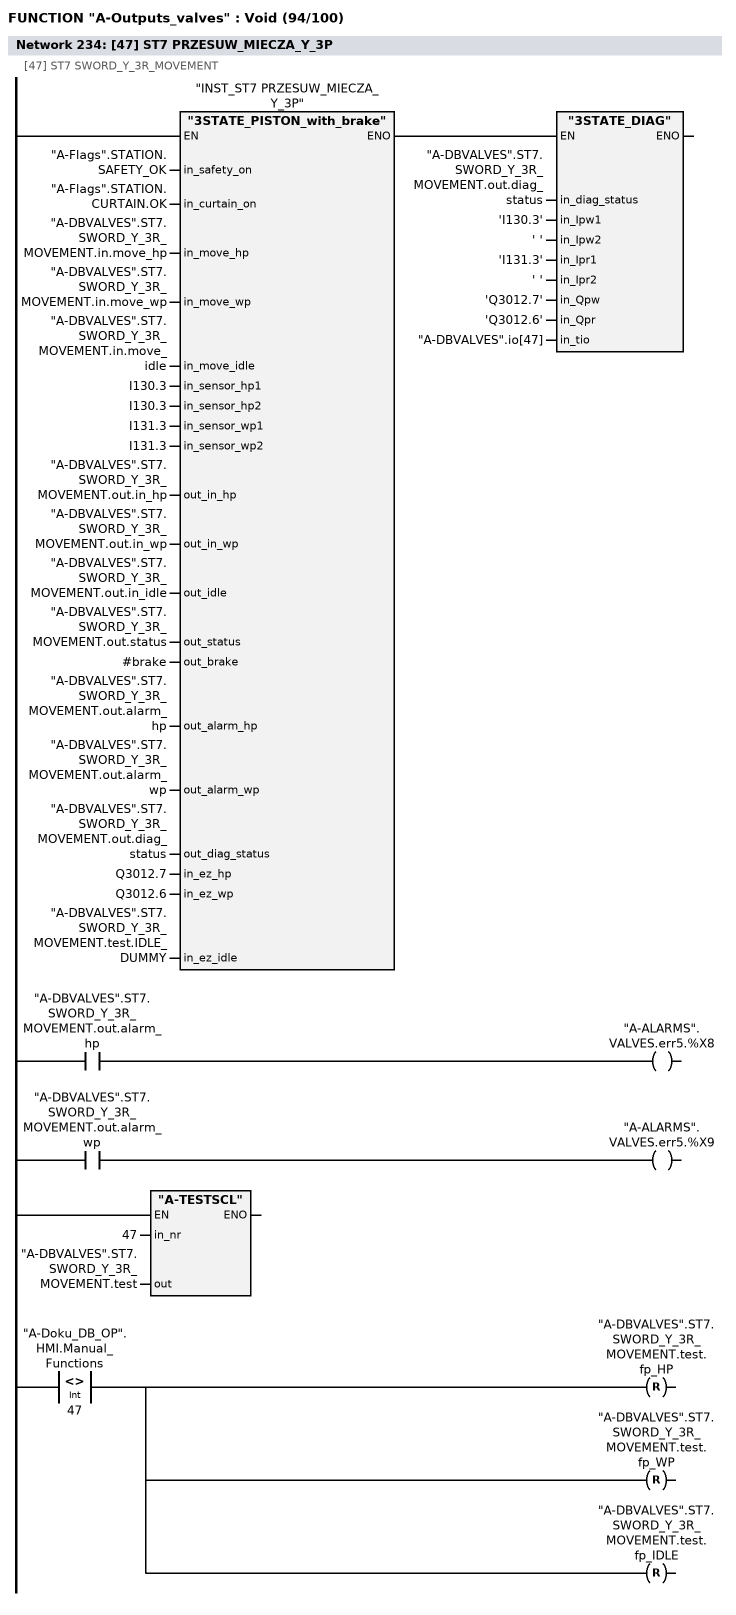
      CALL "3STATE_PISTON_with_brake", "INST_ST7 PRZESUW_MIECZA_Y_3P"
      (  in_safety_on                := "A-Flags".STATION.SAFETY_OK ,
         in_curtain_on               := "A-Flags".STATION.CURTAIN.OK ,
         in_move_hp                  := "A-DBVALVES".ST7.SWORD_Y_3R_MOVEMENT.in.move_hp ,
         in_move_wp                  := "A-DBVALVES".ST7.SWORD_Y_3R_MOVEMENT.in.move_wp ,
         in_move_idle                := "A-DBVALVES".ST7.SWORD_Y_3R_MOVEMENT.in.move_idle ,
         in_sensor_hp1               := I130.3 ,
         in_sensor_hp2               := I130.3 ,
         in_sensor_wp1               := I131.3 ,
         in_sensor_wp2               := I131.3 ,
         out_in_hp                   := "A-DBVALVES".ST7.SWORD_Y_3R_MOVEMENT.out.in_hp ,
         out_in_wp                   := "A-DBVALVES".ST7.SWORD_Y_3R_MOVEMENT.out.in_wp ,
         out_idle                    := "A-DBVALVES".ST7.SWORD_Y_3R_MOVEMENT.out.in_idle ,
         out_status                  := "A-DBVALVES".ST7.SWORD_Y_3R_MOVEMENT.out.status ,
         out_brake                   := #brake ,
         out_alarm_hp                := "A-DBVALVES".ST7.SWORD_Y_3R_MOVEMENT.out.alarm_hp ,
         out_alarm_wp                := "A-DBVALVES".ST7.SWORD_Y_3R_MOVEMENT.out.alarm_wp ,
         out_diag_status             := "A-DBVALVES".ST7.SWORD_Y_3R_MOVEMENT.out.diag_status ,
         in_ez_hp                    := Q3012.7 ,
         in_ez_wp                    := Q3012.6 ,
         in_ez_idle                  := "A-DBVALVES".ST7.SWORD_Y_3R_MOVEMENT.test.IDLE_DUMMY
      );

      CALL "3STATE_DIAG"
      (  in_diag_status              := "A-DBVALVES".ST7.SWORD_Y_3R_MOVEMENT.out.diag_status ,
         in_Ipw1                     := 'I130.3' ,
         in_Ipw2                     := ' ' ,
         in_Ipr1                     := 'I131.3' ,
         in_Ipr2                     := ' ' ,
         in_Qpw                      := 'Q3012.7' ,
         in_Qpr                      := 'Q3012.6' ,
         in_tio                      := "A-DBVALVES".io[47]
      );

      A "A-DBVALVES".ST7.SWORD_Y_3R_MOVEMENT.out.alarm_hp;
      = "A-ALARMS".VALVES.err5.%X8;

      A "A-DBVALVES".ST7.SWORD_Y_3R_MOVEMENT.out.alarm_wp;
      = "A-ALARMS".VALVES.err5.%X9;

      CALL "A-TESTSCL"
      (  in_nr                       := 47 ,
         out                         := "A-DBVALVES".ST7.SWORD_Y_3R_MOVEMENT.test
      );

      A(;
      L "A-Doku_DB_OP".HMI.Manual_Functions;
      L 47;
      <>I;
      );
      R "A-DBVALVES".ST7.SWORD_Y_3R_MOVEMENT.test.fp_HP;
      R "A-DBVALVES".ST7.SWORD_Y_3R_MOVEMENT.test.fp_WP;
      R "A-DBVALVES".ST7.SWORD_Y_3R_MOVEMENT.test.fp_IDLE;
NETWORK
TITLE = -

NETWORK
TITLE = [48] ST7 MIECZ_3P - HP
//[48] ST7 SWORD_3R - HP
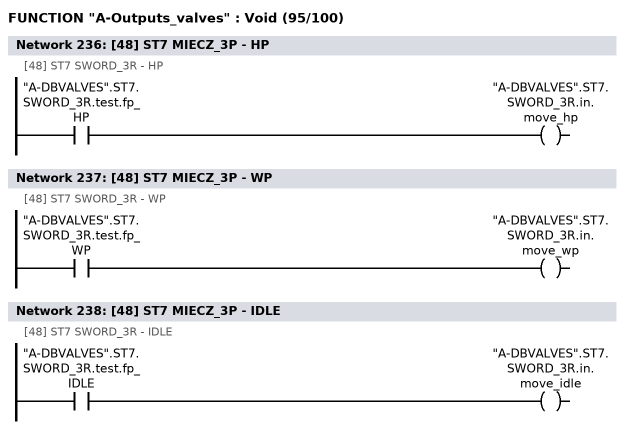
      O "A-DBVALVES".ST7.SWORD_3R.test.fp_HP;
//    O     "A-Flags".STATION.IN_HP_STEP
      = "A-DBVALVES".ST7.SWORD_3R.in.move_hp;
NETWORK
TITLE = [48] ST7 MIECZ_3P - WP
//[48] ST7 SWORD_3R - WP
      O "A-DBVALVES".ST7.SWORD_3R.test.fp_WP;
      = "A-DBVALVES".ST7.SWORD_3R.in.move_wp;
NETWORK
TITLE = [48] ST7 MIECZ_3P - IDLE
//[48] ST7 SWORD_3R - IDLE
      O "A-DBVALVES".ST7.SWORD_3R.test.fp_IDLE;
      = "A-DBVALVES".ST7.SWORD_3R.in.move_idle;
NETWORK
TITLE = [48] ST7 MIECZ_3P
//[48] ST7 SWORD_3R
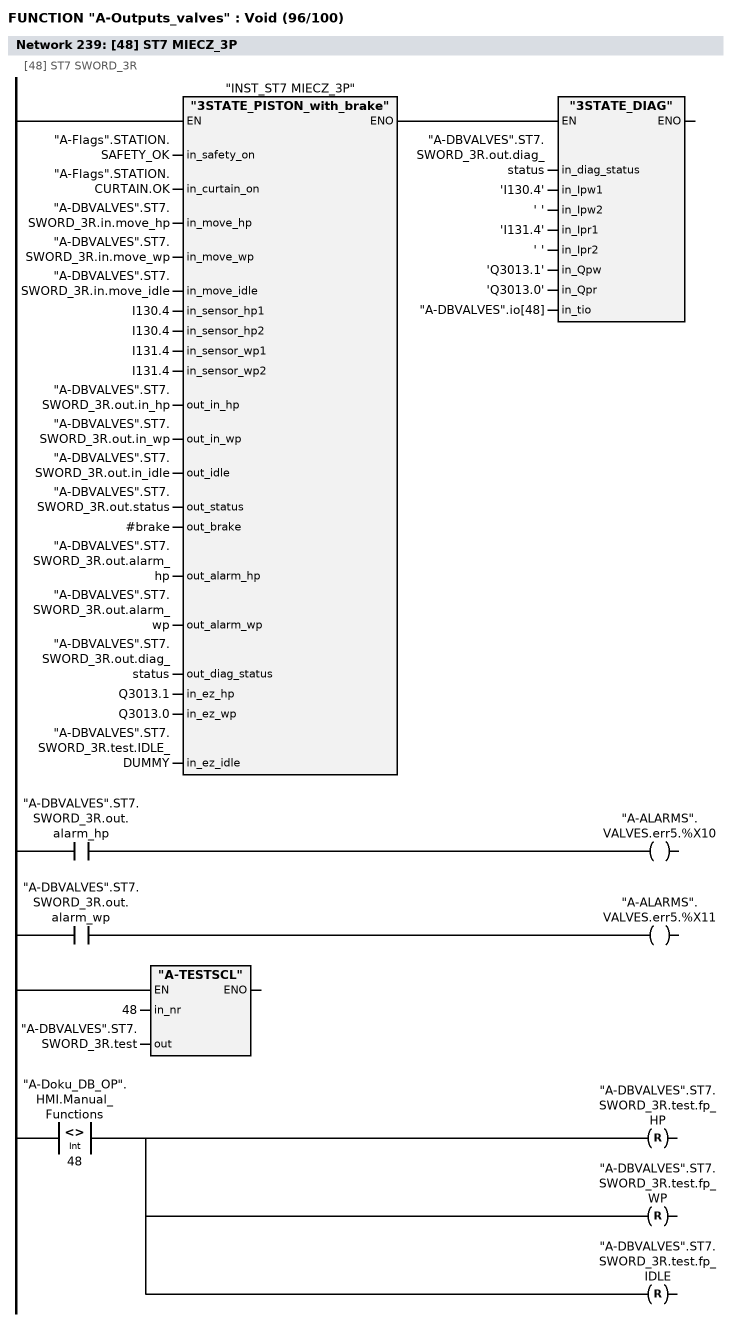
      CALL "3STATE_PISTON_with_brake", "INST_ST7 MIECZ_3P"
      (  in_safety_on                := "A-Flags".STATION.SAFETY_OK ,
         in_curtain_on               := "A-Flags".STATION.CURTAIN.OK ,
         in_move_hp                  := "A-DBVALVES".ST7.SWORD_3R.in.move_hp ,
         in_move_wp                  := "A-DBVALVES".ST7.SWORD_3R.in.move_wp ,
         in_move_idle                := "A-DBVALVES".ST7.SWORD_3R.in.move_idle ,
         in_sensor_hp1               := I130.4 ,
         in_sensor_hp2               := I130.4 ,
         in_sensor_wp1               := I131.4 ,
         in_sensor_wp2               := I131.4 ,
         out_in_hp                   := "A-DBVALVES".ST7.SWORD_3R.out.in_hp ,
         out_in_wp                   := "A-DBVALVES".ST7.SWORD_3R.out.in_wp ,
         out_idle                    := "A-DBVALVES".ST7.SWORD_3R.out.in_idle ,
         out_status                  := "A-DBVALVES".ST7.SWORD_3R.out.status ,
         out_brake                   := #brake ,
         out_alarm_hp                := "A-DBVALVES".ST7.SWORD_3R.out.alarm_hp ,
         out_alarm_wp                := "A-DBVALVES".ST7.SWORD_3R.out.alarm_wp ,
         out_diag_status             := "A-DBVALVES".ST7.SWORD_3R.out.diag_status ,
         in_ez_hp                    := Q3013.1 ,
         in_ez_wp                    := Q3013.0 ,
         in_ez_idle                  := "A-DBVALVES".ST7.SWORD_3R.test.IDLE_DUMMY
      );

      CALL "3STATE_DIAG"
      (  in_diag_status              := "A-DBVALVES".ST7.SWORD_3R.out.diag_status ,
         in_Ipw1                     := 'I130.4' ,
         in_Ipw2                     := ' ' ,
         in_Ipr1                     := 'I131.4' ,
         in_Ipr2                     := ' ' ,
         in_Qpw                      := 'Q3013.1' ,
         in_Qpr                      := 'Q3013.0' ,
         in_tio                      := "A-DBVALVES".io[48]
      );

      A "A-DBVALVES".ST7.SWORD_3R.out.alarm_hp;
      = "A-ALARMS".VALVES.err5.%X10;

      A "A-DBVALVES".ST7.SWORD_3R.out.alarm_wp;
      = "A-ALARMS".VALVES.err5.%X11;

      CALL "A-TESTSCL"
      (  in_nr                       := 48 ,
         out                         := "A-DBVALVES".ST7.SWORD_3R.test
      );

      A(;
      L "A-Doku_DB_OP".HMI.Manual_Functions;
      L 48;
      <>I;
      );
      R "A-DBVALVES".ST7.SWORD_3R.test.fp_HP;
      R "A-DBVALVES".ST7.SWORD_3R.test.fp_WP;
      R "A-DBVALVES".ST7.SWORD_3R.test.fp_IDLE;
NETWORK
TITLE = -

NETWORK
TITLE = [49] ST7 WYSUW_GRZEBIENIA - HP
//[49] ST7 COMB_SLIDE_OUT - HP
